RoboDK station: kr30 cnc 070119 wat.rdk

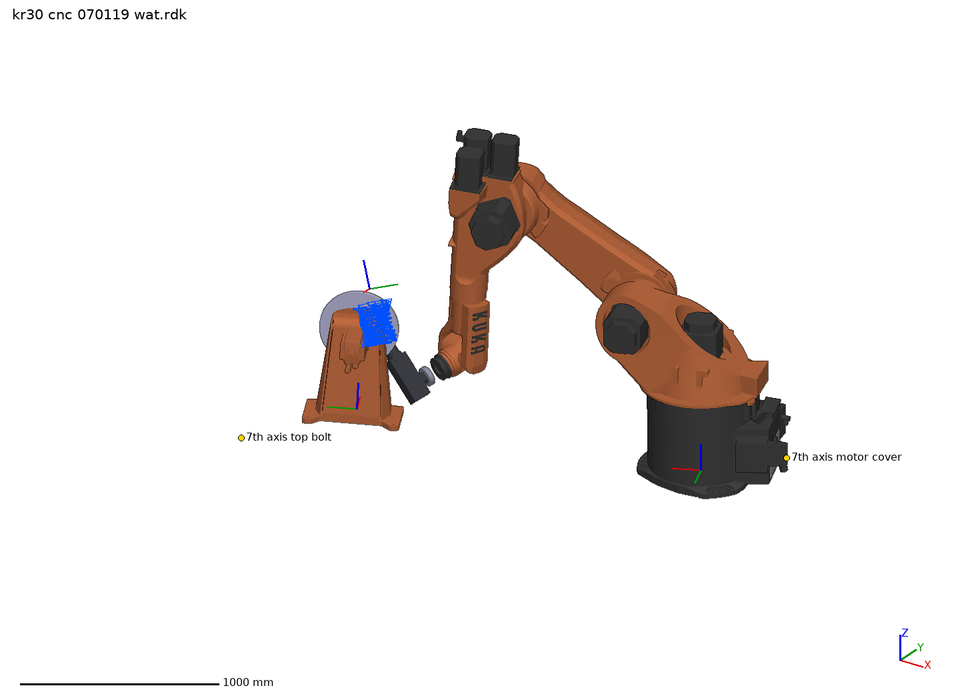
[picture v0: the station drawn from its stored meshes, robots at their saved joint values, targets as dots, program paths as lines]
Station kr30 cnc 070119 wat. Poses are relative to the parent item; angles as X-Y-Z fixed-axis rotations.
  - frame KUKA KR 30 HA Base at (1535.48, 628.29, -1072.61) mm, rotated rx 0 ry 0 rz -156.31 deg
    - robot KUKA KR 30 HA: 6 axes, payload 30 kg, reach 2033 mm, repeatability 0.05 mm, weight 665 kg
        modified DH rows (alpha deg, a mm, theta deg, d mm): 0, 0, 0, 815; -90, 350, 0, 0; 0, 850, -90, 0; -90, 145, 0, 820; 90, 0, 0, 0; -90, 0, 180, 170
        joint limits [-185, -135, -120, -350, -119, -350] to [185, 35, 158, 350, 119, 350]; home [0, -90, 90, 0, 0, 0]; saved at [4.145, -35.537, 122.295, 231.17, 72.258, -40.379]
      - tool 1/2" End Mill TCP, TCP at (337.71, -2.2, 160.57) mm, rotated rx 0 ry 90 rz 0 deg, size 415.8 x 102 x 153.6 mm
    - target 7th axis top bolt (joint target) at (1966.13, 1947.63, 927.26) mm, rotated rx -179.2 ry 6.72 rz -171.11 deg; joints [-17.018, -71.525, 110.046, 168.711, 45.865, -170.331, 883.939] of KUKA KR 30 HA
    - target 7th axis motor cover (joint target) at (-417, -111.35, 57.2) mm, rotated rx -135.46 ry -1.69 rz -48.75 deg; joints [-33.388, -54.543, 96.086, 147.711, 45.276, -113.831, 883.939] of KUKA KR 30 HA
  - frame KUKA KP1 MD250 Base at (172.34, -439.05, -684.5) mm, rotated rx 2 ry 0.52 rz 120.23 deg
    - robot KUKA KP1 MD250: 1 axes, payload 250 kg
        modified DH rows (alpha deg, a mm, theta deg, d mm): 0, 0, 0, 0
        base shift (70, 10, 428) mm, rotated rx 0 ry 90 rz -2 deg
        joint limits [-3600] to [3600]; home [0]; saved at [143.741]
      - frame Frame 2 at (0, 0, 440) mm, rotated rx 0 ry 70 rz 20 deg
  - machining project Machining Settings: C:/Users/liqui/OneDrive/Desktop/suffering.apt | rotz(5) | rotz(80)
  - program Machining (7499 instructions, listed below)
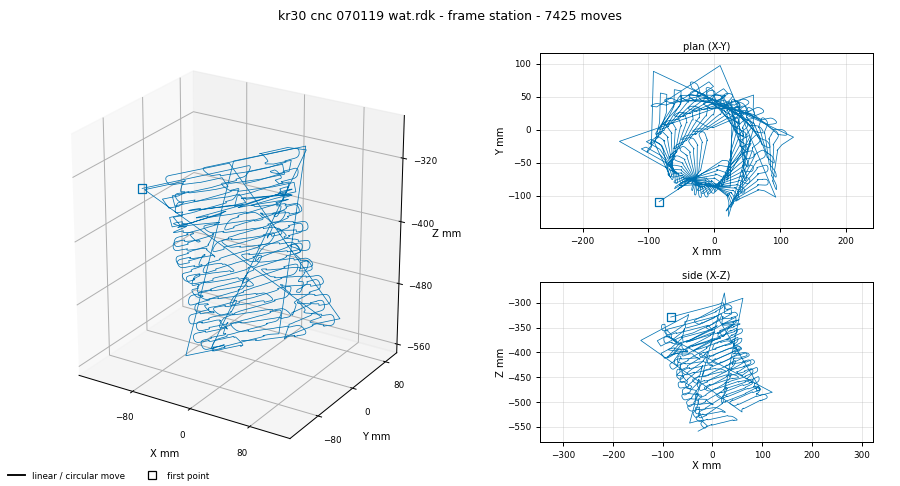
[picture p0: tool path of kr30 cnc 070119 wat.rdk in frame station, 7425 of 7425 moves have a stored position in this frame; points joined in program order, loops and branches not executed]

--- program Machining (robot KUKA KR 30 HA) ---
  Smooth(1)
  Set Ref.: Frame 2
  Set Tool: 1/2" End Mill TCP
  Show 1/2" End Mill TCP
  Print: /'1001'
  Print: /''
  Print: /'Flow1'
  Set speed (1000.0 mm/s)
  Set speed (1000.0 mm/s)
  MoveJ 1 to (78.89, -86.74, -80.36) mm, rotated rx 43.39 ry 15.84 rz 65.61 deg; joints [-0.88, -16.778, 83.729, 155.098, 93.568, 24.647, 178.286]
  MoveL 2 to (78.89, -86.74, -80.36) mm, rotated rx 43.39 ry 15.84 rz 65.61 deg; joints [-0.88, -16.778, 83.729, 155.098, 93.568, 24.647, 178.286]
  MoveL 3 to (78.89, -86.74, -80.36) mm, rotated rx 43.39 ry 15.84 rz 65.61 deg; joints [-0.88, -16.778, 83.729, 155.098, 93.568, 24.647, 178.286]
  Set speed (1000.0 mm/s)
  MoveL 4 to (74.98, -42.03, -80.36) mm, rotated rx 43.39 ry 15.84 rz 65.61 deg; joints [-0.656, -17.28, 87.376, 155.184, 96.389, 23.245, 178.286]
  Set speed (100.0 mm/s)
  MoveL 5 to (68.64, 30.46, -80.36) mm, rotated rx 43.39 ry 15.84 rz 65.61 deg; joints [-0.269, -17.729, 92.84, 155.219, 100.893, 21.011, 178.286]
  MoveL 6 to (68.93, 30.9, -80.36) mm, rotated rx 43.39 ry 15.84 rz 65.61 deg; joints [-0.278, -17.739, 92.882, 155.208, 100.923, 21, 178.286]
  MoveL 7 to (69.23, 31.46, -80.26) mm, rotated rx 43.39 ry 15.84 rz 65.61 deg; joints [-0.286, -17.755, 92.94, 155.197, 100.961, 20.984, 178.286]
  MoveL 8 to (69.53, 31.97, -80.21) mm, rotated rx 43.39 ry 15.84 rz 65.61 deg; joints [-0.294, -17.769, 92.99, 155.187, 100.995, 20.971, 178.286]
  MoveL 9 to (69.83, 32.46, -80.19) mm, rotated rx 43.39 ry 15.84 rz 65.61 deg; joints [-0.303, -17.781, 93.037, 155.176, 101.028, 20.958, 178.286]
  MoveL 10 to (71.83, 35.53, -80.19) mm, rotated rx 43.39 ry 15.84 rz 65.61 deg; joints [-0.366, -17.848, 93.327, 155.099, 101.237, 20.877, 178.286]
  MoveL 11 to (72.67, 36.71, -80.27) mm, rotated rx 43.39 ry 15.84 rz 65.61 deg; joints [-0.394, -17.87, 93.435, 155.066, 101.317, 20.846, 178.286]
  MoveL 12 to (73.47, 37.59, -80.54) mm, rotated rx 43.39 ry 15.84 rz 65.61 deg; joints [-0.423, -17.878, 93.508, 155.033, 101.379, 20.825, 178.286]
  MoveL 13 to (74.21, 38.18, -80.98) mm, rotated rx 43.39 ry 15.84 rz 65.61 deg; joints [-0.455, -17.872, 93.546, 155.001, 101.422, 20.814, 178.286]
  MoveL 14 to (74.56, 38.36, -81.27) mm, rotated rx 43.39 ry 15.84 rz 65.61 deg; joints [-0.471, -17.864, 93.551, 154.985, 101.437, 20.811, 178.286]
  MoveL 15 to (74.9, 38.47, -81.61) mm, rotated rx 43.39 ry 15.84 rz 65.61 deg; joints [-0.487, -17.852, 93.549, 154.969, 101.446, 20.811, 178.286]
  MoveL 16 to (75.55, 38.46, -82.4) mm, rotated rx 43.39 ry 15.84 rz 65.61 deg; joints [-0.521, -17.819, 93.517, 154.937, 101.452, 20.818, 178.286]
  MoveL 17 to (76.14, 38.15, -83.38) mm, rotated rx 43.39 ry 15.84 rz 65.61 deg; joints [-0.557, -17.771, 93.45, 154.906, 101.438, 20.835, 178.286]
  MoveL 18 to (77.19, 36.65, -85.86) mm, rotated rx 43.39 ry 15.84 rz 65.61 deg; joints [-0.633, -17.635, 93.212, 154.845, 101.354, 20.896, 178.286]
  MoveL 19 to (77.76, 34.51, -88.35) mm, rotated rx 43.39 ry 15.84 rz 65.61 deg; joints [-0.693, -17.483, 92.911, 154.802, 101.225, 20.975, 178.286]
  MoveL 20 to (77.59, 32.28, -90.12) mm, rotated rx 43.39 ry 15.84 rz 65.61 deg; joints [-0.717, -17.356, 92.626, 154.793, 101.085, 21.049, 178.286]
  MoveL 21 to (77.22, 31.13, -90.74) mm, rotated rx 43.39 ry 15.84 rz 65.61 deg; joints [-0.715, -17.301, 92.489, 154.801, 101.01, 21.084, 178.286]
  MoveL 22 to (76.67, 29.97, -91.19) mm, rotated rx 43.39 ry 15.84 rz 65.61 deg; joints [-0.705, -17.253, 92.356, 154.818, 100.933, 21.118, 178.286]
  MoveL 23 to (75.02, 27.57, -91.54) mm, rotated rx 43.39 ry 15.84 rz 65.61 deg; joints [-0.657, -17.175, 92.103, 154.876, 100.769, 21.183, 178.286]
  MoveL 24 to (73.01, 25.14, -91.55) mm, rotated rx 43.39 ry 15.84 rz 65.61 deg; joints [-0.593, -17.109, 91.858, 154.95, 100.6, 21.244, 178.286]
  MoveL 25 to (72.71, 24.76, -91.57) mm, rotated rx 43.39 ry 15.84 rz 65.61 deg; joints [-0.583, -17.098, 91.819, 154.96, 100.573, 21.254, 178.286]
  MoveL 26 to (72.43, 24.39, -91.61) mm, rotated rx 43.39 ry 15.84 rz 65.61 deg; joints [-0.575, -17.086, 91.78, 154.97, 100.548, 21.264, 178.286]
  MoveL 27 to (72.2, 24.04, -91.67) mm, rotated rx 43.39 ry 15.84 rz 65.61 deg; joints [-0.569, -17.074, 91.743, 154.978, 100.524, 21.273, 178.286]
  MoveL 28 to (71.94, 23.68, -91.72) mm, rotated rx 43.39 ry 15.84 rz 65.61 deg; joints [-0.561, -17.062, 91.704, 154.987, 100.499, 21.283, 178.286]
  MoveL 29 to (71.6, 23.25, -91.75) mm, rotated rx 43.39 ry 15.84 rz 65.61 deg; joints [-0.551, -17.049, 91.66, 154.999, 100.469, 21.294, 178.286]
  MoveL 30 to (71.2, 22.74, -91.78) mm, rotated rx 43.39 ry 15.84 rz 65.61 deg; joints [-0.539, -17.034, 91.606, 155.013, 100.434, 21.307, 178.286]
  MoveL 31 to (70.87, 22.29, -91.84) mm, rotated rx 43.39 ry 15.84 rz 65.61 deg; joints [-0.529, -17.019, 91.558, 155.025, 100.402, 21.319, 178.286]
  MoveL 32 to (70.62, 21.92, -91.92) mm, rotated rx 43.39 ry 15.84 rz 65.61 deg; joints [-0.522, -17.005, 91.517, 155.033, 100.377, 21.329, 178.286]
  MoveL 33 to (70.37, 21.56, -91.97) mm, rotated rx 43.39 ry 15.84 rz 65.61 deg; joints [-0.515, -16.993, 91.479, 155.042, 100.352, 21.339, 178.286]
  MoveL 34 to (70.07, 21.19, -91.99) mm, rotated rx 43.39 ry 15.84 rz 65.61 deg; joints [-0.506, -16.982, 91.44, 155.052, 100.326, 21.348, 178.286]
  MoveL 35 to (69.74, 20.78, -91.99) mm, rotated rx 43.39 ry 15.84 rz 65.61 deg; joints [-0.495, -16.971, 91.4, 155.064, 100.298, 21.358, 178.286]
  MoveL 36 to (69.39, 20.37, -91.99) mm, rotated rx 43.39 ry 15.84 rz 65.61 deg; joints [-0.484, -16.959, 91.357, 155.077, 100.269, 21.369, 178.286]
  MoveL 37 to (69.04, 19.92, -92) mm, rotated rx 43.39 ry 15.84 rz 65.61 deg; joints [-0.473, -16.947, 91.311, 155.09, 100.238, 21.38, 178.286]
  MoveL 38 to (68.64, 19.39, -92.03) mm, rotated rx 43.39 ry 15.84 rz 65.61 deg; joints [-0.461, -16.931, 91.257, 155.104, 100.201, 21.394, 178.286]
  MoveL 39 to (68.32, 18.89, -92.1) mm, rotated rx 43.39 ry 15.84 rz 65.61 deg; joints [-0.451, -16.915, 91.205, 155.115, 100.167, 21.407, 178.286]
  MoveL 40 to (68.09, 18.5, -92.2) mm, rotated rx 43.39 ry 15.84 rz 65.61 deg; joints [-0.446, -16.9, 91.161, 155.122, 100.14, 21.418, 178.286]
  MoveL 41 to (68.08, 18.51, -92.44) mm, rotated rx 43.39 ry 15.84 rz 65.61 deg; joints [-0.449, -16.885, 91.146, 155.12, 100.14, 21.419, 178.286]
  MoveL 42 to (68.22, 18.88, -92.79) mm, rotated rx 43.39 ry 15.84 rz 65.61 deg; joints [-0.458, -16.869, 91.155, 155.109, 100.165, 21.41, 178.286]
  MoveL 43 to (69.04, 19.11, -93.76) mm, rotated rx 43.39 ry 15.84 rz 65.61 deg; joints [-0.499, -16.831, 91.136, 155.07, 100.186, 21.412, 178.286]
  MoveL 44 to (68.82, 16.99, -93.76) mm, rotated rx 43.39 ry 15.84 rz 65.61 deg; joints [-0.497, -16.812, 90.968, 155.083, 100.051, 21.475, 178.286]
  MoveL 45 to (68.62, 14.7, -93.89) mm, rotated rx 43.39 ry 15.84 rz 65.61 deg; joints [-0.497, -16.783, 90.779, 155.095, 99.906, 21.544, 178.286]
  MoveL 46 to (68.41, 12.54, -93.95) mm, rotated rx 43.39 ry 15.84 rz 65.61 deg; joints [-0.495, -16.759, 90.603, 155.108, 99.768, 21.608, 178.286]
  MoveL 47 to (68.21, 10.42, -94.08) mm, rotated rx 43.39 ry 15.84 rz 65.61 deg; joints [-0.495, -16.731, 90.427, 155.118, 99.634, 21.672, 178.286]
  MoveL 48 to (68.01, 8.29, -94.23) mm, rotated rx 43.39 ry 15.84 rz 65.61 deg; joints [-0.496, -16.7, 90.246, 155.128, 99.498, 21.736, 178.286]
  MoveL 49 to (67.81, 6.18, -94.36) mm, rotated rx 43.39 ry 15.84 rz 65.61 deg; joints [-0.495, -16.671, 90.069, 155.139, 99.363, 21.799, 178.286]
  MoveL 50 to (67.61, 4.04, -94.56) mm, rotated rx 43.39 ry 15.84 rz 65.61 deg; joints [-0.496, -16.637, 89.885, 155.149, 99.227, 21.863, 178.286]
  MoveL 51 to (67.4, 1.93, -94.68) mm, rotated rx 43.39 ry 15.84 rz 65.61 deg; joints [-0.496, -16.608, 89.707, 155.159, 99.092, 21.926, 178.286]
  MoveL 52 to (67.19, -0.21, -94.74) mm, rotated rx 43.39 ry 15.84 rz 65.61 deg; joints [-0.494, -16.582, 89.53, 155.171, 98.955, 21.99, 178.286]
  MoveL 53 to (66.97, -2.35, -94.88) mm, rotated rx 43.39 ry 15.84 rz 65.61 deg; joints [-0.494, -16.549, 89.347, 155.181, 98.818, 22.054, 178.286]
  MoveL 54 to (66.75, -4.57, -95.06) mm, rotated rx 43.39 ry 15.84 rz 65.61 deg; joints [-0.494, -16.514, 89.155, 155.191, 98.676, 22.12, 178.286]
  MoveL 55 to (66.52, -6.78, -95.24) mm, rotated rx 43.39 ry 15.84 rz 65.61 deg; joints [-0.493, -16.478, 88.962, 155.201, 98.534, 22.186, 178.286]
  MoveL 56 to (66.32, -8.65, -95.48) mm, rotated rx 43.39 ry 15.84 rz 65.61 deg; joints [-0.494, -16.441, 88.793, 155.209, 98.414, 22.243, 178.286]
  MoveL 57 to (66.04, -11.3, -95.59) mm, rotated rx 43.39 ry 15.84 rz 65.61 deg; joints [-0.492, -16.403, 88.569, 155.222, 98.244, 22.321, 178.286]
  Set speed (1000.0 mm/s)
  MoveL 58 to (69.99, -56.43, -95.59) mm, rotated rx 43.39 ry 15.84 rz 65.61 deg; joints [-0.725, -16.011, 85.023, 155.17, 95.414, 23.724, 178.286]
  Set speed (1000.0 mm/s)
  MoveL 59 to (64.27, -56.93, -107.47) mm, rotated rx 43.39 ry 15.84 rz 65.61 deg; joints [-0.695, -15.1, 83.995, 155.201, 95.303, 23.764, 178.286]
  Set speed (100.0 mm/s)
  MoveL 60 to (61.77, -28.35, -107.47) mm, rotated rx 43.39 ry 15.84 rz 65.61 deg; joints [-0.549, -15.374, 86.276, 155.242, 97.105, 22.872, 178.286]
  MoveL 61 to (62.19, -26.69, -107.23) mm, rotated rx 43.39 ry 15.84 rz 65.61 deg; joints [-0.556, -15.418, 86.441, 155.23, 97.216, 22.823, 178.286]
  MoveL 62 to (62.63, -24.71, -107.16) mm, rotated rx 43.39 ry 15.84 rz 65.61 deg; joints [-0.565, -15.454, 86.62, 155.213, 97.346, 22.766, 178.286]
  MoveL 63 to (63.09, -22.71, -107.02) mm, rotated rx 43.39 ry 15.84 rz 65.61 deg; joints [-0.574, -15.495, 86.805, 155.197, 97.478, 22.707, 178.286]
  MoveL 64 to (63.66, -20.32, -106.88) mm, rotated rx 43.39 ry 15.84 rz 65.61 deg; joints [-0.586, -15.543, 87.025, 155.176, 97.636, 22.638, 178.286]
  MoveL 65 to (64.13, -18.23, -106.88) mm, rotated rx 43.39 ry 15.84 rz 65.61 deg; joints [-0.598, -15.576, 87.207, 155.158, 97.773, 22.578, 178.286]
  MoveL 66 to (64.64, -15.93, -106.72) mm, rotated rx 43.39 ry 15.84 rz 65.61 deg; joints [-0.608, -15.621, 87.417, 155.139, 97.924, 22.511, 178.286]
  MoveL 67 to (65.09, -13.99, -106.54) mm, rotated rx 43.39 ry 15.84 rz 65.61 deg; joints [-0.616, -15.663, 87.599, 155.123, 98.052, 22.454, 178.286]
  MoveL 68 to (65.55, -12, -106.44) mm, rotated rx 43.39 ry 15.84 rz 65.61 deg; joints [-0.626, -15.699, 87.778, 155.105, 98.183, 22.396, 178.286]
  MoveL 69 to (66.01, -9.91, -106.23) mm, rotated rx 43.39 ry 15.84 rz 65.61 deg; joints [-0.634, -15.744, 87.972, 155.089, 98.32, 22.335, 178.286]
  MoveL 70 to (66.47, -7.85, -106.07) mm, rotated rx 43.39 ry 15.84 rz 65.61 deg; joints [-0.643, -15.784, 88.16, 155.072, 98.455, 22.274, 178.286]
  MoveL 71 to (66.93, -5.79, -105.96) mm, rotated rx 43.39 ry 15.84 rz 65.61 deg; joints [-0.653, -15.821, 88.344, 155.054, 98.589, 22.214, 178.286]
  MoveL 72 to (67.38, -3.69, -105.79) mm, rotated rx 43.39 ry 15.84 rz 65.61 deg; joints [-0.661, -15.861, 88.534, 155.036, 98.726, 22.152, 178.286]
  MoveL 73 to (67.83, -1.62, -105.65) mm, rotated rx 43.39 ry 15.84 rz 65.61 deg; joints [-0.67, -15.899, 88.72, 155.018, 98.862, 22.092, 178.286]
  MoveL 74 to (68.31, 0.51, -105.58) mm, rotated rx 43.39 ry 15.84 rz 65.61 deg; joints [-0.681, -15.933, 88.905, 154.999, 99, 22.03, 178.286]
  MoveL 75 to (68.74, 2.6, -105.38) mm, rotated rx 43.39 ry 15.84 rz 65.61 deg; joints [-0.688, -15.974, 89.095, 154.982, 99.136, 21.968, 178.286]
  MoveL 76 to (69.19, 4.67, -105.25) mm, rotated rx 43.39 ry 15.84 rz 65.61 deg; joints [-0.697, -16.009, 89.278, 154.963, 99.271, 21.907, 178.286]
  MoveL 77 to (69.64, 6.79, -105.13) mm, rotated rx 43.39 ry 15.84 rz 65.61 deg; joints [-0.706, -16.045, 89.464, 154.944, 99.408, 21.845, 178.286]
  MoveL 78 to (69.88, 8.54, -104.92) mm, rotated rx 43.39 ry 15.84 rz 65.61 deg; joints [-0.708, -16.077, 89.621, 154.934, 99.521, 21.792, 178.286]
  MoveL 79 to (69.95, 10.01, -104.57) mm, rotated rx 43.39 ry 15.84 rz 65.61 deg; joints [-0.702, -16.112, 89.76, 154.932, 99.615, 21.746, 178.286]
  MoveL 80 to (69.81, 11.21, -104.04) mm, rotated rx 43.39 ry 15.84 rz 65.61 deg; joints [-0.687, -16.15, 89.882, 154.94, 99.689, 21.706, 178.286]
  MoveL 81 to (69.03, 9.88, -103.19) mm, rotated rx 43.39 ry 15.84 rz 65.61 deg; joints [-0.652, -16.174, 89.813, 154.979, 99.6, 21.737, 178.286]
  MoveL 82 to (69.37, 10.61, -103.19) mm, rotated rx 43.39 ry 15.84 rz 65.61 deg; joints [-0.662, -16.188, 89.879, 154.966, 99.649, 21.717, 178.286]
  MoveL 83 to (69.73, 11.22, -103.19) mm, rotated rx 43.39 ry 15.84 rz 65.61 deg; joints [-0.673, -16.202, 89.937, 154.953, 99.69, 21.701, 178.286]
  MoveL 84 to (70.13, 11.71, -103.18) mm, rotated rx 43.39 ry 15.84 rz 65.61 deg; joints [-0.685, -16.216, 89.988, 154.939, 99.725, 21.688, 178.286]
  MoveL 85 to (70.58, 12.21, -103.16) mm, rotated rx 43.39 ry 15.84 rz 65.61 deg; joints [-0.7, -16.232, 90.041, 154.923, 99.76, 21.676, 178.286]
  MoveL 86 to (71.11, 12.75, -103.13) mm, rotated rx 43.39 ry 15.84 rz 65.61 deg; joints [-0.716, -16.252, 90.102, 154.904, 99.799, 21.663, 178.286]
  MoveL 87 to (72.63, 14.2, -103.13) mm, rotated rx 43.39 ry 15.84 rz 65.61 deg; joints [-0.766, -16.301, 90.26, 154.851, 99.904, 21.628, 178.286]
  MoveL 88 to (72.95, 14.51, -103.11) mm, rotated rx 43.39 ry 15.84 rz 65.61 deg; joints [-0.776, -16.313, 90.295, 154.84, 99.926, 21.621, 178.286]
  MoveL 89 to (73.71, 15.23, -103.11) mm, rotated rx 43.39 ry 15.84 rz 65.61 deg; joints [-0.801, -16.337, 90.374, 154.813, 99.978, 21.603, 178.286]
  MoveL 90 to (74.07, 15.58, -103.1) mm, rotated rx 43.39 ry 15.84 rz 65.61 deg; joints [-0.813, -16.349, 90.412, 154.8, 100.003, 21.595, 178.286]
  MoveL 91 to (74.42, 15.92, -103.08) mm, rotated rx 43.39 ry 15.84 rz 65.61 deg; joints [-0.824, -16.362, 90.45, 154.788, 100.028, 21.587, 178.286]
  MoveL 92 to (74.75, 16.27, -103.05) mm, rotated rx 43.39 ry 15.84 rz 65.61 deg; joints [-0.834, -16.375, 90.489, 154.777, 100.053, 21.578, 178.286]
  MoveL 93 to (75.04, 16.6, -102.99) mm, rotated rx 43.39 ry 15.84 rz 65.61 deg; joints [-0.842, -16.388, 90.527, 154.767, 100.076, 21.57, 178.286]
  MoveL 94 to (75.36, 16.94, -102.96) mm, rotated rx 43.39 ry 15.84 rz 65.61 deg; joints [-0.852, -16.401, 90.566, 154.756, 100.1, 21.561, 178.286]
  MoveL 95 to (75.71, 17.29, -102.94) mm, rotated rx 43.39 ry 15.84 rz 65.61 deg; joints [-0.864, -16.413, 90.604, 154.744, 100.125, 21.552, 178.286]
  MoveL 96 to (76.08, 17.64, -102.93) mm, rotated rx 43.39 ry 15.84 rz 65.61 deg; joints [-0.875, -16.425, 90.643, 154.731, 100.151, 21.544, 178.286]
  MoveL 97 to (76.43, 17.99, -102.91) mm, rotated rx 43.39 ry 15.84 rz 65.61 deg; joints [-0.887, -16.438, 90.682, 154.719, 100.176, 21.535, 178.286]
  MoveL 98 to (76.76, 18.34, -102.87) mm, rotated rx 43.39 ry 15.84 rz 65.61 deg; joints [-0.897, -16.451, 90.721, 154.707, 100.2, 21.527, 178.286]
  MoveL 99 to (77.04, 18.67, -102.82) mm, rotated rx 43.39 ry 15.84 rz 65.61 deg; joints [-0.905, -16.464, 90.758, 154.698, 100.223, 21.518, 178.286]
  MoveL 100 to (77.34, 19.01, -102.76) mm, rotated rx 43.39 ry 15.84 rz 65.61 deg; joints [-0.914, -16.477, 90.797, 154.688, 100.248, 21.509, 178.286]
  MoveL 101 to (78.34, 20.05, -102.68) mm, rotated rx 43.39 ry 15.84 rz 65.61 deg; joints [-0.945, -16.514, 90.912, 154.653, 100.321, 21.483, 178.286]
  MoveL 102 to (79.25, 20.79, -102.81) mm, rotated rx 43.39 ry 15.84 rz 65.61 deg; joints [-0.978, -16.534, 90.988, 154.619, 100.376, 21.467, 178.286]
  MoveL 103 to (80.08, 21.23, -103.15) mm, rotated rx 43.39 ry 15.84 rz 65.61 deg; joints [-1.01, -16.537, 91.025, 154.586, 100.41, 21.46, 178.286]
  MoveL 104 to (80.47, 21.34, -103.39) mm, rotated rx 43.39 ry 15.84 rz 65.61 deg; joints [-1.027, -16.532, 91.029, 154.57, 100.42, 21.46, 178.286]
  MoveL 105 to (80.83, 21.38, -103.69) mm, rotated rx 43.39 ry 15.84 rz 65.61 deg; joints [-1.044, -16.523, 91.023, 154.554, 100.425, 21.463, 178.286]
  MoveL 106 to (81.5, 21.23, -104.45) mm, rotated rx 43.39 ry 15.84 rz 65.61 deg; joints [-1.078, -16.491, 90.982, 154.524, 100.421, 21.475, 178.286]
  MoveL 107 to (82.09, 20.78, -105.42) mm, rotated rx 43.39 ry 15.84 rz 65.61 deg; joints [-1.113, -16.442, 90.902, 154.494, 100.397, 21.497, 178.286]
  MoveL 108 to (83.02, 19, -107.98) mm, rotated rx 43.39 ry 15.84 rz 65.61 deg; joints [-1.184, -16.293, 90.626, 154.438, 100.291, 21.57, 178.286]
  MoveL 109 to (83.37, 16.68, -110.59) mm, rotated rx 43.39 ry 15.84 rz 65.61 deg; joints [-1.237, -16.122, 90.287, 154.403, 100.145, 21.657, 178.286]
  MoveL 110 to (83.23, 15.57, -111.62) mm, rotated rx 43.39 ry 15.84 rz 65.61 deg; joints [-1.249, -16.046, 90.129, 154.399, 100.073, 21.696, 178.286]
  MoveL 111 to (82.89, 14.48, -112.46) mm, rotated rx 43.39 ry 15.84 rz 65.61 deg; joints [-1.25, -15.977, 89.98, 154.403, 100.001, 21.732, 178.286]
  MoveL 112 to (82.34, 13.43, -113.11) mm, rotated rx 43.39 ry 15.84 rz 65.61 deg; joints [-1.242, -15.914, 89.839, 154.417, 99.929, 21.764, 178.286]
  MoveL 113 to (81.58, 12.41, -113.58) mm, rotated rx 43.39 ry 15.84 rz 65.61 deg; joints [-1.224, -15.859, 89.707, 154.439, 99.858, 21.793, 178.286]
  MoveL 114 to (80.61, 11.42, -113.86) mm, rotated rx 43.39 ry 15.84 rz 65.61 deg; joints [-1.197, -15.809, 89.582, 154.47, 99.787, 21.819, 178.286]
  MoveL 115 to (79.44, 10.46, -113.95) mm, rotated rx 43.39 ry 15.84 rz 65.61 deg; joints [-1.159, -15.766, 89.466, 154.51, 99.716, 21.841, 178.286]
  MoveL 116 to (76.9, 8.59, -113.96) mm, rotated rx 43.39 ry 15.84 rz 65.61 deg; joints [-1.075, -15.688, 89.242, 154.597, 99.575, 21.883, 178.286]
  MoveL 117 to (76.46, 8.25, -113.97) mm, rotated rx 43.39 ry 15.84 rz 65.61 deg; joints [-1.061, -15.673, 89.201, 154.612, 99.55, 21.89, 178.286]
  MoveL 118 to (75.97, 7.86, -114.01) mm, rotated rx 43.39 ry 15.84 rz 65.61 deg; joints [-1.045, -15.655, 89.154, 154.629, 99.521, 21.899, 178.286]
  MoveL 119 to (75.4, 7.36, -114.1) mm, rotated rx 43.39 ry 15.84 rz 65.61 deg; joints [-1.028, -15.631, 89.091, 154.647, 99.484, 21.911, 178.286]
  MoveL 120 to (74.92, 6.97, -114.14) mm, rotated rx 43.39 ry 15.84 rz 65.61 deg; joints [-1.012, -15.613, 89.043, 154.664, 99.455, 21.92, 178.286]
  MoveL 121 to (74.49, 6.64, -114.15) mm, rotated rx 43.39 ry 15.84 rz 65.61 deg; joints [-0.998, -15.599, 89.003, 154.678, 99.43, 21.928, 178.286]
  MoveL 122 to (74.08, 6.34, -114.16) mm, rotated rx 43.39 ry 15.84 rz 65.61 deg; joints [-0.985, -15.585, 88.967, 154.692, 99.407, 21.935, 178.286]
  MoveL 123 to (73.72, 6.05, -114.18) mm, rotated rx 43.39 ry 15.84 rz 65.61 deg; joints [-0.974, -15.573, 88.932, 154.704, 99.386, 21.941, 178.286]
  MoveL 124 to (72.07, 4.82, -114.18) mm, rotated rx 43.39 ry 15.84 rz 65.61 deg; joints [-0.919, -15.521, 88.785, 154.76, 99.293, 21.968, 178.286]
  MoveL 125 to (71.67, 4.5, -114.22) mm, rotated rx 43.39 ry 15.84 rz 65.61 deg; joints [-0.907, -15.506, 88.745, 154.774, 99.269, 21.975, 178.286]
  MoveL 126 to (71.32, 4.19, -114.27) mm, rotated rx 43.39 ry 15.84 rz 65.61 deg; joints [-0.896, -15.491, 88.706, 154.785, 99.246, 21.983, 178.286]
  MoveL 127 to (70.98, 3.88, -114.34) mm, rotated rx 43.39 ry 15.84 rz 65.61 deg; joints [-0.886, -15.475, 88.666, 154.796, 99.223, 21.991, 178.286]
  MoveL 128 to (70.64, 3.53, -114.4) mm, rotated rx 43.39 ry 15.84 rz 65.61 deg; joints [-0.876, -15.46, 88.624, 154.807, 99.198, 22, 178.286]
  MoveL 129 to (70.27, 3.12, -114.44) mm, rotated rx 43.39 ry 15.84 rz 65.61 deg; joints [-0.865, -15.445, 88.578, 154.82, 99.169, 22.01, 178.286]
  MoveL 130 to (69.89, 2.57, -114.44) mm, rotated rx 43.39 ry 15.84 rz 65.61 deg; joints [-0.853, -15.43, 88.522, 154.833, 99.13, 22.024, 178.286]
  MoveL 131 to (69.51, 1.89, -114.45) mm, rotated rx 43.39 ry 15.84 rz 65.61 deg; joints [-0.841, -15.415, 88.458, 154.847, 99.084, 22.043, 178.286]
  MoveL 132 to (71.15, 2.93, -116) mm, rotated rx 43.39 ry 15.84 rz 65.61 deg; joints [-0.917, -15.367, 88.486, 154.773, 99.162, 22.03, 178.286]
  MoveL 133 to (70.38, 0.7, -116.13) mm, rotated rx 43.39 ry 15.84 rz 65.61 deg; joints [-0.897, -15.321, 88.279, 154.802, 99.014, 22.094, 178.286]
  MoveL 134 to (69.65, -1.41, -116.24) mm, rotated rx 43.39 ry 15.84 rz 65.61 deg; joints [-0.877, -15.278, 88.083, 154.83, 98.873, 22.154, 178.286]
  MoveL 135 to (68.95, -3.46, -116.4) mm, rotated rx 43.39 ry 15.84 rz 65.61 deg; joints [-0.86, -15.232, 87.89, 154.856, 98.737, 22.213, 178.286]
  MoveL 136 to (68.25, -5.47, -116.51) mm, rotated rx 43.39 ry 15.84 rz 65.61 deg; joints [-0.842, -15.19, 87.702, 154.882, 98.603, 22.271, 178.286]
  MoveL 137 to (67.55, -7.49, -116.62) mm, rotated rx 43.39 ry 15.84 rz 65.61 deg; joints [-0.824, -15.147, 87.513, 154.908, 98.468, 22.329, 178.286]
  MoveL 138 to (66.86, -9.51, -116.84) mm, rotated rx 43.39 ry 15.84 rz 65.61 deg; joints [-0.807, -15.097, 87.316, 154.932, 98.333, 22.387, 178.286]
  MoveL 139 to (66.16, -11.53, -117.07) mm, rotated rx 43.39 ry 15.84 rz 65.61 deg; joints [-0.791, -15.047, 87.119, 154.956, 98.198, 22.445, 178.286]
  MoveL 140 to (65.45, -13.54, -117.18) mm, rotated rx 43.39 ry 15.84 rz 65.61 deg; joints [-0.773, -15.002, 86.928, 154.981, 98.063, 22.503, 178.286]
  MoveL 141 to (64.73, -15.55, -117.18) mm, rotated rx 43.39 ry 15.84 rz 65.61 deg; joints [-0.753, -14.964, 86.745, 155.008, 97.929, 22.559, 178.286]
  MoveL 142 to (64.02, -17.56, -117.29) mm, rotated rx 43.39 ry 15.84 rz 65.61 deg; joints [-0.734, -14.919, 86.553, 155.033, 97.794, 22.616, 178.286]
  MoveL 143 to (63.29, -19.6, -117.5) mm, rotated rx 43.39 ry 15.84 rz 65.61 deg; joints [-0.717, -14.867, 86.352, 155.058, 97.656, 22.675, 178.286]
  MoveL 144 to (62.62, -21.5, -117.67) mm, rotated rx 43.39 ry 15.84 rz 65.61 deg; joints [-0.701, -14.819, 86.166, 155.08, 97.528, 22.729, 178.286]
  MoveL 145 to (61.99, -23.25, -117.89) mm, rotated rx 43.39 ry 15.84 rz 65.61 deg; joints [-0.686, -14.772, 85.99, 155.1, 97.41, 22.779, 178.286]
  MoveL 146 to (61.33, -25.1, -117.98) mm, rotated rx 43.39 ry 15.84 rz 65.61 deg; joints [-0.669, -14.729, 85.812, 155.123, 97.285, 22.831, 178.286]
  MoveL 147 to (60.62, -27.07, -117.99) mm, rotated rx 43.39 ry 15.84 rz 65.61 deg; joints [-0.65, -14.689, 85.629, 155.148, 97.152, 22.886, 178.286]
  MoveL 148 to (59.7, -29.61, -118.09) mm, rotated rx 43.39 ry 15.84 rz 65.61 deg; joints [-0.625, -14.631, 85.384, 155.18, 96.98, 22.958, 178.286]
  MoveL 149 to (58.99, -31.52, -118.3) mm, rotated rx 43.39 ry 15.84 rz 65.61 deg; joints [-0.609, -14.578, 85.191, 155.202, 96.85, 23.012, 178.286]
  MoveL 150 to (58.22, -33.58, -118.51) mm, rotated rx 43.39 ry 15.84 rz 65.61 deg; joints [-0.59, -14.522, 84.983, 155.227, 96.709, 23.071, 178.286]
  MoveL 151 to (57.5, -35.47, -118.79) mm, rotated rx 43.39 ry 15.84 rz 65.61 deg; joints [-0.574, -14.464, 84.784, 155.248, 96.58, 23.125, 178.286]
  MoveL 152 to (56.82, -37.34, -118.92) mm, rotated rx 43.39 ry 15.84 rz 65.61 deg; joints [-0.557, -14.416, 84.599, 155.27, 96.453, 23.178, 178.286]
  MoveL 153 to (56.11, -39.31, -118.94) mm, rotated rx 43.39 ry 15.84 rz 65.61 deg; joints [-0.538, -14.373, 84.412, 155.294, 96.319, 23.233, 178.286]
  MoveL 154 to (55.46, -40.96, -119.17) mm, rotated rx 43.39 ry 15.84 rz 65.61 deg; joints [-0.523, -14.322, 84.238, 155.313, 96.205, 23.279, 178.286]
  Set speed (1000.0 mm/s)
  MoveL 155 to (57.74, -66.91, -119.17) mm, rotated rx 43.39 ry 15.84 rz 65.61 deg; joints [-0.655, -14.043, 82.122, 155.266, 94.556, 24.094, 178.286]
  Set speed (1000.0 mm/s)
  MoveL 156 to (51.22, -67.48, -130.35) mm, rotated rx 43.39 ry 15.84 rz 65.61 deg; joints [-0.591, -13.142, 81.063, 155.33, 94.403, 24.138, 178.286]
  Set speed (100.0 mm/s)
  MoveL 157 to (49.47, -47.39, -130.35) mm, rotated rx 43.39 ry 15.84 rz 65.61 deg; joints [-0.488, -13.368, 82.718, 155.369, 95.685, 23.506, 178.286]
  MoveL 158 to (50.43, -45.49, -130.35) mm, rotated rx 43.39 ry 15.84 rz 65.61 deg; joints [-0.516, -13.418, 82.911, 155.338, 95.819, 23.455, 178.286]
  MoveL 159 to (51.46, -43.51, -130.25) mm, rotated rx 43.39 ry 15.84 rz 65.61 deg; joints [-0.545, -13.476, 83.118, 155.306, 95.959, 23.401, 178.286]
  MoveL 160 to (52.58, -41.44, -129.96) mm, rotated rx 43.39 ry 15.84 rz 65.61 deg; joints [-0.573, -13.55, 83.349, 155.273, 96.106, 23.344, 178.286]
  MoveL 161 to (53.65, -39.46, -129.62) mm, rotated rx 43.39 ry 15.84 rz 65.61 deg; joints [-0.6, -13.624, 83.574, 155.242, 96.247, 23.289, 178.286]
  MoveL 162 to (54.61, -37.63, -129.43) mm, rotated rx 43.39 ry 15.84 rz 65.61 deg; joints [-0.625, -13.684, 83.771, 155.213, 96.376, 23.239, 178.286]
  MoveL 163 to (55.5, -35.9, -129.29) mm, rotated rx 43.39 ry 15.84 rz 65.61 deg; joints [-0.65, -13.736, 83.954, 155.185, 96.498, 23.191, 178.286]
  MoveL 164 to (56.44, -34.07, -129.24) mm, rotated rx 43.39 ry 15.84 rz 65.61 deg; joints [-0.676, -13.785, 84.14, 155.154, 96.625, 23.142, 178.286]
  MoveL 165 to (57.4, -32.17, -129.22) mm, rotated rx 43.39 ry 15.84 rz 65.61 deg; joints [-0.704, -13.834, 84.33, 155.122, 96.758, 23.09, 178.286]
  MoveL 166 to (58.36, -30.28, -129.1) mm, rotated rx 43.39 ry 15.84 rz 65.61 deg; joints [-0.731, -13.887, 84.525, 155.091, 96.89, 23.039, 178.286]
  MoveL 167 to (59.41, -28.24, -128.84) mm, rotated rx 43.39 ry 15.84 rz 65.61 deg; joints [-0.758, -13.954, 84.744, 155.058, 97.032, 22.982, 178.286]
  MoveL 168 to (60.49, -26.1, -128.66) mm, rotated rx 43.39 ry 15.84 rz 65.61 deg; joints [-0.787, -14.017, 84.968, 155.023, 97.181, 22.923, 178.286]
  MoveL 169 to (61.54, -24.01, -128.45) mm, rotated rx 43.39 ry 15.84 rz 65.61 deg; joints [-0.815, -14.079, 85.185, 154.989, 97.326, 22.865, 178.286]
  MoveL 170 to (62.5, -22.11, -128.34) mm, rotated rx 43.39 ry 15.84 rz 65.61 deg; joints [-0.842, -14.131, 85.379, 154.957, 97.458, 22.812, 178.286]
  MoveL 171 to (64.38, -18.33, -128.07) mm, rotated rx 43.39 ry 15.84 rz 65.61 deg; joints [-0.894, -14.236, 85.764, 154.894, 97.719, 22.708, 178.286]
  MoveL 172 to (65.36, -16.38, -128) mm, rotated rx 43.39 ry 15.84 rz 65.61 deg; joints [-0.923, -14.285, 85.957, 154.86, 97.853, 22.654, 178.286]
  MoveL 173 to (66.3, -14.47, -127.78) mm, rotated rx 43.39 ry 15.84 rz 65.61 deg; joints [-0.947, -14.342, 86.156, 154.829, 97.985, 22.6, 178.286]
  MoveL 174 to (67.23, -12.57, -127.62) mm, rotated rx 43.39 ry 15.84 rz 65.61 deg; joints [-0.973, -14.394, 86.348, 154.797, 98.115, 22.547, 178.286]
  MoveL 175 to (68.15, -10.67, -127.44) mm, rotated rx 43.39 ry 15.84 rz 65.61 deg; joints [-0.998, -14.448, 86.542, 154.766, 98.245, 22.494, 178.286]
  MoveL 176 to (69.12, -8.72, -127.34) mm, rotated rx 43.39 ry 15.84 rz 65.61 deg; joints [-1.026, -14.496, 86.734, 154.731, 98.378, 22.44, 178.286]
  MoveL 177 to (70.11, -6.68, -127.22) mm, rotated rx 43.39 ry 15.84 rz 65.61 deg; joints [-1.054, -14.548, 86.936, 154.696, 98.518, 22.383, 178.286]
  MoveL 178 to (70.97, -4.98, -127.16) mm, rotated rx 43.39 ry 15.84 rz 65.61 deg; joints [-1.079, -14.589, 87.102, 154.665, 98.634, 22.336, 178.286]
  MoveL 179 to (70.38, -4.68, -126.27) mm, rotated rx 43.39 ry 15.84 rz 65.61 deg; joints [-1.046, -14.633, 87.167, 154.694, 98.649, 22.318, 178.286]
  MoveL 180 to (70.06, -4.84, -125.86) mm, rotated rx 43.39 ry 15.84 rz 65.61 deg; joints [-1.03, -14.65, 87.173, 154.709, 98.637, 22.318, 178.286]
  MoveL 181 to (69.99, -4.83, -125.58) mm, rotated rx 43.39 ry 15.84 rz 65.61 deg; joints [-1.024, -14.666, 87.19, 154.715, 98.638, 22.315, 178.286]
  MoveL 182 to (70.25, -4.63, -125.46) mm, rotated rx 43.39 ry 15.84 rz 65.61 deg; joints [-1.031, -14.681, 87.222, 154.707, 98.654, 22.31, 178.286]
  MoveL 183 to (70.62, -4.38, -125.4) mm, rotated rx 43.39 ry 15.84 rz 65.61 deg; joints [-1.042, -14.697, 87.258, 154.696, 98.673, 22.305, 178.286]
  MoveL 184 to (71.1, -4.08, -125.37) mm, rotated rx 43.39 ry 15.84 rz 65.61 deg; joints [-1.057, -14.714, 87.299, 154.68, 98.697, 22.298, 178.286]
  MoveL 185 to (71.69, -3.72, -125.33) mm, rotated rx 43.39 ry 15.84 rz 65.61 deg; joints [-1.076, -14.735, 87.349, 154.661, 98.726, 22.291, 178.286]
  MoveL 186 to (72.24, -3.4, -125.31) mm, rotated rx 43.39 ry 15.84 rz 65.61 deg; joints [-1.094, -14.753, 87.394, 154.643, 98.751, 22.285, 178.286]
  MoveL 187 to (72.69, -3.14, -125.31) mm, rotated rx 43.39 ry 15.84 rz 65.61 deg; joints [-1.109, -14.767, 87.428, 154.628, 98.772, 22.28, 178.286]
  MoveL 188 to (73.12, -2.89, -125.29) mm, rotated rx 43.39 ry 15.84 rz 65.61 deg; joints [-1.123, -14.781, 87.462, 154.614, 98.792, 22.275, 178.286]
  MoveL 189 to (73.99, -2.34, -125.21) mm, rotated rx 43.39 ry 15.84 rz 65.61 deg; joints [-1.151, -14.814, 87.539, 154.586, 98.836, 22.263, 178.286]
  MoveL 190 to (74.47, -2.03, -125.16) mm, rotated rx 43.39 ry 15.84 rz 65.61 deg; joints [-1.166, -14.831, 87.581, 154.57, 98.859, 22.257, 178.286]
  MoveL 191 to (74.88, -1.74, -125.09) mm, rotated rx 43.39 ry 15.84 rz 65.61 deg; joints [-1.178, -14.849, 87.622, 154.557, 98.882, 22.25, 178.286]
  MoveL 192 to (75.26, -1.47, -125.02) mm, rotated rx 43.39 ry 15.84 rz 65.61 deg; joints [-1.19, -14.866, 87.66, 154.545, 98.903, 22.244, 178.286]
  MoveL 193 to (75.65, -1.22, -124.96) mm, rotated rx 43.39 ry 15.84 rz 65.61 deg; joints [-1.202, -14.881, 87.696, 154.533, 98.923, 22.238, 178.286]
  MoveL 194 to (76.06, -0.96, -124.93) mm, rotated rx 43.39 ry 15.84 rz 65.61 deg; joints [-1.215, -14.896, 87.732, 154.52, 98.943, 22.233, 178.286]
  MoveL 195 to (76.51, -0.69, -124.91) mm, rotated rx 43.39 ry 15.84 rz 65.61 deg; joints [-1.23, -14.911, 87.768, 154.505, 98.964, 22.227, 178.286]
  MoveL 196 to (79.7, 1.1, -124.91) mm, rotated rx 43.39 ry 15.84 rz 65.61 deg; joints [-1.336, -15.008, 88.008, 154.398, 99.107, 22.193, 178.286]
  MoveL 197 to (81.17, 1.8, -124.93) mm, rotated rx 43.39 ry 15.84 rz 65.61 deg; joints [-1.385, -15.05, 88.107, 154.349, 99.165, 22.181, 178.286]
  MoveL 198 to (81.72, 1.97, -124.96) mm, rotated rx 43.39 ry 15.84 rz 65.61 deg; joints [-1.404, -15.063, 88.135, 154.33, 99.18, 22.18, 178.286]
  MoveL 199 to (82.16, 2.01, -124.99) mm, rotated rx 43.39 ry 15.84 rz 65.61 deg; joints [-1.42, -15.073, 88.15, 154.316, 99.187, 22.182, 178.286]
  MoveL 200 to (82.5, 1.96, -125.03) mm, rotated rx 43.39 ry 15.84 rz 65.61 deg; joints [-1.432, -15.078, 88.153, 154.305, 99.187, 22.186, 178.286]
  MoveL 201 to (82.63, 1.89, -125.06) mm, rotated rx 43.39 ry 15.84 rz 65.61 deg; joints [-1.437, -15.08, 88.151, 154.3, 99.184, 22.189, 178.286]
  MoveL 202 to (82.74, 1.81, -125.08) mm, rotated rx 43.39 ry 15.84 rz 65.61 deg; joints [-1.441, -15.08, 88.146, 154.297, 99.179, 22.193, 178.286]
  MoveL 203 to (82.83, 1.7, -125.11) mm, rotated rx 43.39 ry 15.84 rz 65.61 deg; joints [-1.445, -15.08, 88.139, 154.294, 99.173, 22.197, 178.286]
  MoveL 204 to (82.9, 1.58, -125.14) mm, rotated rx 43.39 ry 15.84 rz 65.61 deg; joints [-1.448, -15.079, 88.129, 154.292, 99.166, 22.201, 178.286]
  MoveL 205 to (82.98, 1.27, -125.2) mm, rotated rx 43.39 ry 15.84 rz 65.61 deg; joints [-1.452, -15.075, 88.103, 154.29, 99.147, 22.212, 178.286]
  MoveL 206 to (82.93, 0.48, -125.33) mm, rotated rx 43.39 ry 15.84 rz 65.61 deg; joints [-1.453, -15.059, 88.031, 154.292, 99.097, 22.237, 178.286]
  MoveL 207 to (82.67, -0.5, -125.47) mm, rotated rx 43.39 ry 15.84 rz 65.61 deg; joints [-1.448, -15.035, 87.938, 154.302, 99.033, 22.266, 178.286]
  MoveL 208 to (81.78, -2.66, -125.74) mm, rotated rx 43.39 ry 15.84 rz 65.61 deg; joints [-1.425, -14.977, 87.722, 154.334, 98.888, 22.329, 178.286]
  MoveL 209 to (80.71, -4.82, -125.98) mm, rotated rx 43.39 ry 15.84 rz 65.61 deg; joints [-1.395, -14.916, 87.502, 154.372, 98.741, 22.391, 178.286]
  MoveL 210 to (56.48, -53.07, -131.06) mm, rotated rx 43.39 ry 15.84 rz 65.61 deg; joints [-0.742, -13.437, 82.427, 155.155, 95.397, 23.739, 178.286]
  MoveL 211 to (54.76, -56.49, -131.42) mm, rotated rx 43.39 ry 15.84 rz 65.61 deg; joints [-0.697, -13.322, 82.052, 155.205, 95.154, 23.834, 178.286]
  MoveL 212 to (52.92, -59.76, -131.84) mm, rotated rx 43.39 ry 15.84 rz 65.61 deg; joints [-0.649, -13.201, 81.681, 155.258, 94.92, 23.923, 178.286]
  MoveL 213 to (51.96, -60.9, -132.05) mm, rotated rx 43.39 ry 15.84 rz 65.61 deg; joints [-0.623, -13.146, 81.536, 155.285, 94.833, 23.953, 178.286]
  MoveL 214 to (51.51, -61.2, -132.15) mm, rotated rx 43.39 ry 15.84 rz 65.61 deg; joints [-0.61, -13.124, 81.487, 155.298, 94.808, 23.959, 178.286]
  MoveL 215 to (51.29, -61.27, -132.19) mm, rotated rx 43.39 ry 15.84 rz 65.61 deg; joints [-0.604, -13.114, 81.471, 155.304, 94.8, 23.96, 178.286]
  MoveL 216 to (51.08, -61.28, -132.23) mm, rotated rx 43.39 ry 15.84 rz 65.61 deg; joints [-0.597, -13.106, 81.46, 155.309, 94.797, 23.959, 178.286]
  MoveL 217 to (50.88, -61.21, -132.27) mm, rotated rx 43.39 ry 15.84 rz 65.61 deg; joints [-0.591, -13.099, 81.456, 155.315, 94.799, 23.955, 178.286]
  MoveL 218 to (50.69, -61.08, -132.3) mm, rotated rx 43.39 ry 15.84 rz 65.61 deg; joints [-0.585, -13.094, 81.459, 155.32, 94.806, 23.95, 178.286]
  MoveL 219 to (50.52, -60.86, -132.33) mm, rotated rx 43.39 ry 15.84 rz 65.61 deg; joints [-0.579, -13.09, 81.469, 155.325, 94.817, 23.942, 178.286]
  MoveL 220 to (50.35, -60.56, -132.36) mm, rotated rx 43.39 ry 15.84 rz 65.61 deg; joints [-0.573, -13.088, 81.487, 155.329, 94.835, 23.932, 178.286]
  MoveL 221 to (49.85, -58.43, -132.41) mm, rotated rx 43.39 ry 15.84 rz 65.61 deg; joints [-0.553, -13.101, 81.65, 155.342, 94.967, 23.862, 178.286]
  MoveL 222 to (49.6, -56.35, -132.41) mm, rotated rx 43.39 ry 15.84 rz 65.61 deg; joints [-0.54, -13.123, 81.819, 155.349, 95.099, 23.796, 178.286]
  MoveL 223 to (49.6, -52.55, -132.45) mm, rotated rx 43.39 ry 15.84 rz 65.61 deg; joints [-0.532, -13.171, 82.139, 155.345, 95.345, 23.68, 178.286]
  MoveL 224 to (50.37, -49.09, -132.56) mm, rotated rx 43.39 ry 15.84 rz 65.61 deg; joints [-0.551, -13.229, 82.45, 155.318, 95.578, 23.58, 178.286]
  MoveL 225 to (53.08, -43.68, -132.86) mm, rotated rx 43.39 ry 15.84 rz 65.61 deg; joints [-0.634, -13.35, 82.975, 155.226, 95.957, 23.437, 178.286]
  MoveL 226 to (54.56, -41.83, -132.99) mm, rotated rx 43.39 ry 15.84 rz 65.61 deg; joints [-0.68, -13.404, 83.17, 155.178, 96.092, 23.392, 178.286]
  MoveL 227 to (77.42, -15.64, -134.86) mm, rotated rx 43.39 ry 15.84 rz 65.61 deg; joints [-1.422, -14.168, 85.928, 154.4, 98, 22.759, 178.286]
  MoveL 228 to (79.36, -13.39, -135.02) mm, rotated rx 43.39 ry 15.84 rz 65.61 deg; joints [-1.487, -14.229, 86.158, 154.331, 98.161, 22.704, 178.286]
  MoveL 229 to (81.44, -10.29, -135.26) mm, rotated rx 43.39 ry 15.84 rz 65.61 deg; joints [-1.555, -14.296, 86.453, 154.254, 98.376, 22.623, 178.286]
  MoveL 230 to (81.98, -8.9, -135.4) mm, rotated rx 43.39 ry 15.84 rz 65.61 deg; joints [-1.573, -14.313, 86.57, 154.231, 98.468, 22.584, 178.286]
  MoveL 231 to (82.01, -8.36, -135.47) mm, rotated rx 43.39 ry 15.84 rz 65.61 deg; joints [-1.574, -14.315, 86.61, 154.227, 98.502, 22.567, 178.286]
  MoveL 232 to (81.96, -8.14, -135.51) mm, rotated rx 43.39 ry 15.84 rz 65.61 deg; joints [-1.573, -14.313, 86.623, 154.228, 98.516, 22.56, 178.286]
  MoveL 233 to (81.86, -7.95, -135.54) mm, rotated rx 43.39 ry 15.84 rz 65.61 deg; joints [-1.57, -14.31, 86.632, 154.23, 98.526, 22.554, 178.286]
  MoveL 234 to (81.7, -7.81, -135.58) mm, rotated rx 43.39 ry 15.84 rz 65.61 deg; joints [-1.564, -14.305, 86.636, 154.234, 98.533, 22.549, 178.286]
  MoveL 235 to (81.49, -7.72, -135.61) mm, rotated rx 43.39 ry 15.84 rz 65.61 deg; joints [-1.557, -14.298, 86.634, 154.24, 98.537, 22.545, 178.286]
  MoveL 236 to (81.21, -7.67, -135.64) mm, rotated rx 43.39 ry 15.84 rz 65.61 deg; joints [-1.548, -14.289, 86.627, 154.248, 98.537, 22.542, 178.286]
  MoveL 237 to (80.87, -7.68, -135.68) mm, rotated rx 43.39 ry 15.84 rz 65.61 deg; joints [-1.537, -14.278, 86.613, 154.259, 98.533, 22.54, 178.286]
  MoveL 238 to (78.78, -8.34, -135.8) mm, rotated rx 43.39 ry 15.84 rz 65.61 deg; joints [-1.469, -14.211, 86.486, 154.325, 98.471, 22.547, 178.286]
  MoveL 239 to (78.3, -8.55, -135.82) mm, rotated rx 43.39 ry 15.84 rz 65.61 deg; joints [-1.453, -14.195, 86.454, 154.34, 98.453, 22.55, 178.286]
  MoveL 240 to (77.89, -8.76, -135.87) mm, rotated rx 43.39 ry 15.84 rz 65.61 deg; joints [-1.44, -14.18, 86.421, 154.353, 98.436, 22.554, 178.286]
  MoveL 241 to (77.51, -8.97, -135.94) mm, rotated rx 43.39 ry 15.84 rz 65.61 deg; joints [-1.428, -14.163, 86.386, 154.365, 98.418, 22.558, 178.286]
  MoveL 242 to (77.11, -9.18, -136) mm, rotated rx 43.39 ry 15.84 rz 65.61 deg; joints [-1.416, -14.148, 86.354, 154.378, 98.401, 22.562, 178.286]
  MoveL 243 to (76.7, -9.38, -136.03) mm, rotated rx 43.39 ry 15.84 rz 65.61 deg; joints [-1.403, -14.133, 86.322, 154.391, 98.384, 22.566, 178.286]
  MoveL 244 to (72.36, -11.14, -136.04) mm, rotated rx 43.39 ry 15.84 rz 65.61 deg; joints [-1.258, -14.004, 86.043, 154.532, 98.23, 22.591, 178.286]
  MoveL 245 to (71.95, -11.32, -136.06) mm, rotated rx 43.39 ry 15.84 rz 65.61 deg; joints [-1.245, -13.991, 86.014, 154.545, 98.214, 22.594, 178.286]
  MoveL 246 to (71.51, -11.51, -136.08) mm, rotated rx 43.39 ry 15.84 rz 65.61 deg; joints [-1.231, -13.977, 85.985, 154.559, 98.198, 22.597, 178.286]
  MoveL 247 to (70.55, -11.9, -136.08) mm, rotated rx 43.39 ry 15.84 rz 65.61 deg; joints [-1.199, -13.948, 85.922, 154.59, 98.163, 22.602, 178.286]
  MoveL 248 to (70.03, -12.12, -136.08) mm, rotated rx 43.39 ry 15.84 rz 65.61 deg; joints [-1.182, -13.932, 85.887, 154.607, 98.144, 22.606, 178.286]
  MoveL 249 to (69.48, -12.38, -136.1) mm, rotated rx 43.39 ry 15.84 rz 65.61 deg; joints [-1.164, -13.914, 85.848, 154.624, 98.122, 22.61, 178.286]
  MoveL 250 to (68.9, -12.69, -136.13) mm, rotated rx 43.39 ry 15.84 rz 65.61 deg; joints [-1.145, -13.894, 85.802, 154.643, 98.096, 22.616, 178.286]
  MoveL 251 to (68.36, -13.07, -136.15) mm, rotated rx 43.39 ry 15.84 rz 65.61 deg; joints [-1.128, -13.875, 85.752, 154.661, 98.066, 22.624, 178.286]
  MoveL 252 to (67.85, -13.49, -136.17) mm, rotated rx 43.39 ry 15.84 rz 65.61 deg; joints [-1.112, -13.857, 85.701, 154.677, 98.034, 22.634, 178.286]
  MoveL 253 to (69.02, -12.9, -137.15) mm, rotated rx 43.39 ry 15.84 rz 65.61 deg; joints [-1.164, -13.831, 85.718, 154.627, 98.081, 22.63, 178.286]
  MoveL 254 to (68.56, -14.15, -137.58) mm, rotated rx 43.39 ry 15.84 rz 65.61 deg; joints [-1.156, -13.779, 85.573, 154.64, 97.994, 22.668, 178.286]
  MoveL 255 to (67.92, -15.5, -137.9) mm, rotated rx 43.39 ry 15.84 rz 65.61 deg; joints [-1.141, -13.729, 85.422, 154.66, 97.901, 22.708, 178.286]
  MoveL 256 to (67.08, -16.98, -138.13) mm, rotated rx 43.39 ry 15.84 rz 65.61 deg; joints [-1.119, -13.678, 85.26, 154.686, 97.798, 22.749, 178.286]
  MoveL 257 to (65.93, -18.77, -138.35) mm, rotated rx 43.39 ry 15.84 rz 65.61 deg; joints [-1.086, -13.616, 85.062, 154.724, 97.671, 22.799, 178.286]
  MoveL 258 to (64.75, -20.55, -138.46) mm, rotated rx 43.39 ry 15.84 rz 65.61 deg; joints [-1.052, -13.56, 84.872, 154.763, 97.545, 22.846, 178.286]
  MoveL 259 to (63.57, -22.33, -138.57) mm, rotated rx 43.39 ry 15.84 rz 65.61 deg; joints [-1.017, -13.504, 84.681, 154.802, 97.418, 22.894, 178.286]
  MoveL 260 to (62.4, -24.12, -138.8) mm, rotated rx 43.39 ry 15.84 rz 65.61 deg; joints [-0.984, -13.44, 84.481, 154.839, 97.291, 22.942, 178.286]
  MoveL 261 to (61.22, -25.89, -138.92) mm, rotated rx 43.39 ry 15.84 rz 65.61 deg; joints [-0.949, -13.382, 84.29, 154.878, 97.164, 22.99, 178.286]
  MoveL 262 to (60.04, -27.67, -139.15) mm, rotated rx 43.39 ry 15.84 rz 65.61 deg; joints [-0.917, -13.317, 84.089, 154.915, 97.037, 23.038, 178.286]
  MoveL 263 to (58.85, -29.44, -139.27) mm, rotated rx 43.39 ry 15.84 rz 65.61 deg; joints [-0.882, -13.259, 83.896, 154.954, 96.91, 23.085, 178.286]
  MoveL 264 to (57.66, -31.21, -139.39) mm, rotated rx 43.39 ry 15.84 rz 65.61 deg; joints [-0.847, -13.2, 83.702, 154.992, 96.783, 23.132, 178.286]
  MoveL 265 to (56.47, -32.98, -139.62) mm, rotated rx 43.39 ry 15.84 rz 65.61 deg; joints [-0.814, -13.134, 83.5, 155.029, 96.655, 23.179, 178.286]
  MoveL 266 to (55.32, -34.67, -139.73) mm, rotated rx 43.39 ry 15.84 rz 65.61 deg; joints [-0.781, -13.077, 83.314, 155.065, 96.534, 23.224, 178.286]
  MoveL 267 to (54.19, -36.3, -139.93) mm, rotated rx 43.39 ry 15.84 rz 65.61 deg; joints [-0.749, -13.015, 83.126, 155.1, 96.415, 23.268, 178.286]
  MoveL 268 to (52.87, -38.27, -140.09) mm, rotated rx 43.39 ry 15.84 rz 65.61 deg; joints [-0.711, -12.946, 82.906, 155.141, 96.272, 23.32, 178.286]
  MoveL 269 to (51.31, -40.51, -140.18) mm, rotated rx 43.39 ry 15.84 rz 65.61 deg; joints [-0.666, -12.872, 82.661, 155.19, 96.11, 23.378, 178.286]
  MoveL 270 to (50.15, -42.23, -140.25) mm, rotated rx 43.39 ry 15.84 rz 65.61 deg; joints [-0.632, -12.816, 82.473, 155.227, 95.985, 23.423, 178.286]
  MoveL 271 to (49.07, -43.82, -140.38) mm, rotated rx 43.39 ry 15.84 rz 65.61 deg; joints [-0.601, -12.759, 82.293, 155.26, 95.869, 23.465, 178.286]
  MoveL 272 to (47.95, -45.46, -140.48) mm, rotated rx 43.39 ry 15.84 rz 65.61 deg; joints [-0.569, -12.702, 82.109, 155.294, 95.75, 23.507, 178.286]
  MoveL 273 to (46.84, -47.06, -140.59) mm, rotated rx 43.39 ry 15.84 rz 65.61 deg; joints [-0.537, -12.644, 81.927, 155.328, 95.632, 23.55, 178.286]
  MoveL 274 to (45.68, -48.77, -140.66) mm, rotated rx 43.39 ry 15.84 rz 65.61 deg; joints [-0.504, -12.587, 81.739, 155.364, 95.508, 23.594, 178.286]
  MoveL 275 to (44.42, -50.6, -140.76) mm, rotated rx 43.39 ry 15.84 rz 65.61 deg; joints [-0.467, -12.523, 81.532, 155.402, 95.373, 23.641, 178.286]
  MoveL 276 to (43.02, -52.56, -141.02) mm, rotated rx 43.39 ry 15.84 rz 65.61 deg; joints [-0.429, -12.442, 81.298, 155.442, 95.228, 23.693, 178.286]
  MoveL 277 to (42.2, -54.64, -142.01) mm, rotated rx 43.39 ry 15.84 rz 65.61 deg; joints [-0.42, -12.328, 81.021, 155.457, 95.078, 23.758, 178.286]
  MoveL 278 to (42.21, -53.5, -142.49) mm, rotated rx 43.39 ry 15.84 rz 65.61 deg; joints [-0.424, -12.313, 81.083, 155.45, 95.15, 23.727, 178.286]
  MoveL 279 to (42.22, -52.9, -142.8) mm, rotated rx 43.39 ry 15.84 rz 65.61 deg; joints [-0.427, -12.301, 81.112, 155.446, 95.187, 23.711, 178.286]
  MoveL 280 to (42.21, -52.8, -142.95) mm, rotated rx 43.39 ry 15.84 rz 65.61 deg; joints [-0.429, -12.292, 81.11, 155.444, 95.193, 23.709, 178.286]
  MoveL 281 to (42.21, -53.15, -142.99) mm, rotated rx 43.39 ry 15.84 rz 65.61 deg; joints [-0.43, -12.285, 81.077, 155.444, 95.17, 23.72, 178.286]
  MoveL 282 to (42.2, -53.61, -143.01) mm, rotated rx 43.39 ry 15.84 rz 65.61 deg; joints [-0.431, -12.278, 81.036, 155.445, 95.139, 23.734, 178.286]
  MoveL 283 to (42.17, -54.09, -143.04) mm, rotated rx 43.39 ry 15.84 rz 65.61 deg; joints [-0.432, -12.268, 80.992, 155.445, 95.108, 23.749, 178.286]
  MoveL 284 to (42.14, -54.54, -143.1) mm, rotated rx 43.39 ry 15.84 rz 65.61 deg; joints [-0.432, -12.257, 80.948, 155.446, 95.078, 23.763, 178.286]
  MoveL 285 to (42.11, -55, -143.14) mm, rotated rx 43.39 ry 15.84 rz 65.61 deg; joints [-0.433, -12.248, 80.904, 155.447, 95.047, 23.777, 178.286]
  MoveL 286 to (42.1, -55.49, -143.16) mm, rotated rx 43.39 ry 15.84 rz 65.61 deg; joints [-0.434, -12.239, 80.86, 155.447, 95.015, 23.792, 178.286]
  MoveL 287 to (42.08, -58.11, -143.16) mm, rotated rx 43.39 ry 15.84 rz 65.61 deg; joints [-0.439, -12.203, 80.635, 155.449, 94.844, 23.873, 178.286]
  MoveL 288 to (42.07, -58.57, -143.18) mm, rotated rx 43.39 ry 15.84 rz 65.61 deg; joints [-0.44, -12.195, 80.594, 155.449, 94.814, 23.887, 178.286]
  MoveL 289 to (42.04, -58.96, -143.21) mm, rotated rx 43.39 ry 15.84 rz 65.61 deg; joints [-0.441, -12.186, 80.557, 155.45, 94.788, 23.899, 178.286]
  MoveL 290 to (42.03, -59.42, -143.24) mm, rotated rx 43.39 ry 15.84 rz 65.61 deg; joints [-0.441, -12.178, 80.515, 155.45, 94.758, 23.913, 178.286]
  MoveL 291 to (42.01, -60.01, -143.26) mm, rotated rx 43.39 ry 15.84 rz 65.61 deg; joints [-0.443, -12.168, 80.462, 155.451, 94.719, 23.932, 178.286]
  MoveL 292 to (41.97, -60.74, -143.31) mm, rotated rx 43.39 ry 15.84 rz 65.61 deg; joints [-0.443, -12.153, 80.394, 155.452, 94.671, 23.954, 178.286]
  MoveL 293 to (41.94, -61.35, -143.34) mm, rotated rx 43.39 ry 15.84 rz 65.61 deg; joints [-0.444, -12.142, 80.338, 155.452, 94.63, 23.973, 178.286]
  MoveL 294 to (41.94, -61.89, -143.34) mm, rotated rx 43.39 ry 15.84 rz 65.61 deg; joints [-0.446, -12.134, 80.291, 155.453, 94.595, 23.99, 178.286]
  MoveL 295 to (41.93, -63.46, -143.34) mm, rotated rx 43.39 ry 15.84 rz 65.61 deg; joints [-0.449, -12.111, 80.155, 155.454, 94.492, 24.038, 178.286]
  MoveL 296 to (41.62, -66.35, -143.68) mm, rotated rx 43.39 ry 15.84 rz 65.61 deg; joints [-0.45, -12.038, 79.867, 155.46, 94.297, 24.128, 178.286]
  MoveL 297 to (41.25, -67.6, -144.11) mm, rotated rx 43.39 ry 15.84 rz 65.61 deg; joints [-0.446, -11.982, 79.714, 155.466, 94.209, 24.167, 178.286]
  MoveL 298 to (40.73, -68.7, -144.71) mm, rotated rx 43.39 ry 15.84 rz 65.61 deg; joints [-0.439, -11.912, 79.556, 155.475, 94.127, 24.202, 178.286]
  MoveL 299 to (39.25, -70.49, -146.42) mm, rotated rx 43.39 ry 15.84 rz 65.61 deg; joints [-0.418, -11.734, 79.221, 155.499, 93.981, 24.259, 178.286]
  MoveL 300 to (37.18, -71.72, -148.82) mm, rotated rx 43.39 ry 15.84 rz 65.61 deg; joints [-0.385, -11.502, 78.862, 155.532, 93.859, 24.301, 178.286]
  MoveL 301 to (35.17, -72.16, -151.21) mm, rotated rx 43.39 ry 15.84 rz 65.61 deg; joints [-0.352, -11.284, 78.573, 155.563, 93.79, 24.318, 178.286]
  MoveL 302 to (34.43, -72, -152.16) mm, rotated rx 43.39 ry 15.84 rz 65.61 deg; joints [-0.34, -11.205, 78.491, 155.574, 93.785, 24.315, 178.286]
  MoveL 303 to (33.86, -71.58, -152.93) mm, rotated rx 43.39 ry 15.84 rz 65.61 deg; joints [-0.33, -11.146, 78.45, 155.582, 93.8, 24.304, 178.286]
  MoveL 304 to (33.63, -71.27, -153.25) mm, rotated rx 43.39 ry 15.84 rz 65.61 deg; joints [-0.327, -11.123, 78.445, 155.585, 93.815, 24.296, 178.286]
  MoveL 305 to (33.46, -70.9, -153.52) mm, rotated rx 43.39 ry 15.84 rz 65.61 deg; joints [-0.324, -11.106, 78.45, 155.587, 93.836, 24.285, 178.286]
  MoveL 306 to (33.23, -69.97, -153.95) mm, rotated rx 43.39 ry 15.84 rz 65.61 deg; joints [-0.32, -11.086, 78.493, 155.589, 93.892, 24.258, 178.286]
  MoveL 307 to (33.18, -68.78, -154.21) mm, rotated rx 43.39 ry 15.84 rz 65.61 deg; joints [-0.319, -11.087, 78.577, 155.587, 93.968, 24.223, 178.286]
  MoveL 308 to (33.3, -67.34, -154.29) mm, rotated rx 43.39 ry 15.84 rz 65.61 deg; joints [-0.321, -11.106, 78.702, 155.583, 94.064, 24.18, 178.286]
  MoveL 309 to (33.37, -66.82, -154.29) mm, rotated rx 43.39 ry 15.84 rz 65.61 deg; joints [-0.322, -11.116, 78.75, 155.581, 94.099, 24.165, 178.286]
  MoveL 310 to (33.47, -66.39, -154.24) mm, rotated rx 43.39 ry 15.84 rz 65.61 deg; joints [-0.323, -11.129, 78.795, 155.579, 94.129, 24.152, 178.286]
  MoveL 311 to (33.57, -65.97, -154.18) mm, rotated rx 43.39 ry 15.84 rz 65.61 deg; joints [-0.325, -11.142, 78.84, 155.576, 94.159, 24.139, 178.286]
  MoveL 312 to (33.66, -65.5, -154.14) mm, rotated rx 43.39 ry 15.84 rz 65.61 deg; joints [-0.326, -11.154, 78.887, 155.574, 94.191, 24.125, 178.286]
  MoveL 313 to (33.73, -65.01, -154.12) mm, rotated rx 43.39 ry 15.84 rz 65.61 deg; joints [-0.327, -11.164, 78.934, 155.572, 94.224, 24.11, 178.286]
  MoveL 314 to (33.81, -64.48, -154.12) mm, rotated rx 43.39 ry 15.84 rz 65.61 deg; joints [-0.328, -11.175, 78.984, 155.57, 94.26, 24.094, 178.286]
  MoveL 315 to (33.88, -63.96, -154.12) mm, rotated rx 43.39 ry 15.84 rz 65.61 deg; joints [-0.329, -11.184, 79.032, 155.567, 94.295, 24.079, 178.286]
  MoveL 316 to (33.93, -63.46, -154.13) mm, rotated rx 43.39 ry 15.84 rz 65.61 deg; joints [-0.33, -11.192, 79.077, 155.566, 94.329, 24.064, 178.286]
  MoveL 317 to (33.99, -62.97, -154.15) mm, rotated rx 43.39 ry 15.84 rz 65.61 deg; joints [-0.331, -11.2, 79.121, 155.564, 94.362, 24.049, 178.286]
  MoveL 318 to (34.06, -62.51, -154.13) mm, rotated rx 43.39 ry 15.84 rz 65.61 deg; joints [-0.332, -11.21, 79.165, 155.562, 94.393, 24.035, 178.286]
  MoveL 319 to (34.14, -62.05, -154.09) mm, rotated rx 43.39 ry 15.84 rz 65.61 deg; joints [-0.333, -11.222, 79.211, 155.56, 94.424, 24.021, 178.286]
  MoveL 320 to (34.25, -61.52, -154.04) mm, rotated rx 43.39 ry 15.84 rz 65.61 deg; joints [-0.335, -11.236, 79.265, 155.557, 94.461, 24.005, 178.286]
  MoveL 321 to (34.39, -60.83, -153.98) mm, rotated rx 43.39 ry 15.84 rz 65.61 deg; joints [-0.337, -11.253, 79.334, 155.553, 94.508, 23.985, 178.286]
  MoveL 322 to (34.49, -60.19, -153.96) mm, rotated rx 43.39 ry 15.84 rz 65.61 deg; joints [-0.339, -11.267, 79.395, 155.55, 94.552, 23.966, 178.286]
  MoveL 323 to (34.84, -57.6, -153.96) mm, rotated rx 43.39 ry 15.84 rz 65.61 deg; joints [-0.344, -11.313, 79.632, 155.539, 94.726, 23.888, 178.286]
  MoveL 324 to (34.94, -56.98, -153.92) mm, rotated rx 43.39 ry 15.84 rz 65.61 deg; joints [-0.345, -11.327, 79.692, 155.536, 94.768, 23.87, 178.286]
  MoveL 325 to (35.04, -56.43, -153.86) mm, rotated rx 43.39 ry 15.84 rz 65.61 deg; joints [-0.346, -11.341, 79.747, 155.534, 94.806, 23.853, 178.286]
  MoveL 326 to (35.08, -56.23, -153.71) mm, rotated rx 43.39 ry 15.84 rz 65.61 deg; joints [-0.345, -11.355, 79.777, 155.534, 94.82, 23.846, 178.286]
  MoveL 327 to (35.06, -56.35, -153.45) mm, rotated rx 43.39 ry 15.84 rz 65.61 deg; joints [-0.341, -11.37, 79.785, 155.538, 94.814, 23.847, 178.286]
  MoveL 328 to (34.97, -56.79, -153.05) mm, rotated rx 43.39 ry 15.84 rz 65.61 deg; joints [-0.334, -11.387, 79.773, 155.545, 94.786, 23.857, 178.286]
  MoveL 329 to (35.98, -56.6, -152.24) mm, rotated rx 43.39 ry 15.84 rz 65.61 deg; joints [-0.356, -11.47, 79.885, 155.525, 94.816, 23.852, 178.286]
  MoveL 330 to (37.33, -55.16, -152.02) mm, rotated rx 43.39 ry 15.84 rz 65.61 deg; joints [-0.394, -11.541, 80.074, 155.486, 94.929, 23.816, 178.286]
  MoveL 331 to (38.68, -53.68, -151.87) mm, rotated rx 43.39 ry 15.84 rz 65.61 deg; joints [-0.433, -11.608, 80.261, 155.447, 95.044, 23.779, 178.286]
  MoveL 332 to (40.06, -52.15, -151.71) mm, rotated rx 43.39 ry 15.84 rz 65.61 deg; joints [-0.473, -11.676, 80.452, 155.406, 95.162, 23.741, 178.286]
  MoveL 333 to (41.33, -50.77, -151.42) mm, rotated rx 43.39 ry 15.84 rz 65.61 deg; joints [-0.508, -11.748, 80.637, 155.37, 95.269, 23.705, 178.286]
  MoveL 334 to (42.75, -49.2, -151.23) mm, rotated rx 43.39 ry 15.84 rz 65.61 deg; joints [-0.548, -11.82, 80.834, 155.329, 95.39, 23.666, 178.286]
  MoveL 335 to (44.23, -47.56, -151.05) mm, rotated rx 43.39 ry 15.84 rz 65.61 deg; joints [-0.591, -11.893, 81.039, 155.285, 95.516, 23.625, 178.286]
  MoveL 336 to (45.73, -45.89, -150.96) mm, rotated rx 43.39 ry 15.84 rz 65.61 deg; joints [-0.636, -11.961, 81.239, 155.239, 95.643, 23.583, 178.286]
  MoveL 337 to (47.54, -43.85, -150.87) mm, rotated rx 43.39 ry 15.84 rz 65.61 deg; joints [-0.69, -12.041, 81.481, 155.183, 95.797, 23.533, 178.286]
  MoveL 338 to (48.84, -42.38, -150.77) mm, rotated rx 43.39 ry 15.84 rz 65.61 deg; joints [-0.729, -12.101, 81.657, 155.144, 95.908, 23.496, 178.286]
  MoveL 339 to (50.05, -41.01, -150.55) mm, rotated rx 43.39 ry 15.84 rz 65.61 deg; joints [-0.763, -12.164, 81.83, 155.108, 96.012, 23.461, 178.286]
  MoveL 340 to (51.38, -39.5, -150.36) mm, rotated rx 43.39 ry 15.84 rz 65.61 deg; joints [-0.802, -12.231, 82.016, 155.067, 96.127, 23.422, 178.286]
  MoveL 341 to (52.79, -37.9, -150.24) mm, rotated rx 43.39 ry 15.84 rz 65.61 deg; joints [-0.844, -12.296, 82.207, 155.024, 96.247, 23.382, 178.286]
  MoveL 342 to (54.18, -36.3, -150.06) mm, rotated rx 43.39 ry 15.84 rz 65.61 deg; joints [-0.884, -12.363, 82.4, 154.981, 96.367, 23.341, 178.286]
  MoveL 343 to (55.57, -34.71, -149.94) mm, rotated rx 43.39 ry 15.84 rz 65.61 deg; joints [-0.926, -12.427, 82.588, 154.937, 96.486, 23.301, 178.286]
  MoveL 344 to (57, -33.07, -149.76) mm, rotated rx 43.39 ry 15.84 rz 65.61 deg; joints [-0.968, -12.495, 82.786, 154.893, 96.609, 23.259, 178.286]
  MoveL 345 to (58.4, -31.46, -149.64) mm, rotated rx 43.39 ry 15.84 rz 65.61 deg; joints [-1.01, -12.558, 82.974, 154.849, 96.728, 23.218, 178.286]
  MoveL 346 to (59.79, -29.83, -149.41) mm, rotated rx 43.39 ry 15.84 rz 65.61 deg; joints [-1.05, -12.628, 83.172, 154.806, 96.849, 23.175, 178.286]
  MoveL 347 to (61.19, -28.22, -149.3) mm, rotated rx 43.39 ry 15.84 rz 65.61 deg; joints [-1.092, -12.69, 83.359, 154.761, 96.969, 23.134, 178.286]
  MoveL 348 to (62.58, -26.6, -149.18) mm, rotated rx 43.39 ry 15.84 rz 65.61 deg; joints [-1.134, -12.752, 83.547, 154.717, 97.088, 23.093, 178.286]
  MoveL 349 to (63.96, -24.97, -148.96) mm, rotated rx 43.39 ry 15.84 rz 65.61 deg; joints [-1.174, -12.82, 83.742, 154.673, 97.209, 23.05, 178.286]
  MoveL 350 to (65.17, -23.46, -148.76) mm, rotated rx 43.39 ry 15.84 rz 65.61 deg; joints [-1.209, -12.881, 83.92, 154.635, 97.32, 23.01, 178.286]
  MoveL 351 to (66.22, -22.04, -148.46) mm, rotated rx 43.39 ry 15.84 rz 65.61 deg; joints [-1.238, -12.942, 84.09, 154.603, 97.423, 22.971, 178.286]
  MoveL 352 to (67.13, -20.68, -148.06) mm, rotated rx 43.39 ry 15.84 rz 65.61 deg; joints [-1.261, -13.006, 84.259, 154.576, 97.521, 22.932, 178.286]
  MoveL 353 to (65.81, -21.39, -147.13) mm, rotated rx 43.39 ry 15.84 rz 65.61 deg; joints [-1.205, -13.024, 84.225, 154.63, 97.466, 22.939, 178.286]
  MoveL 354 to (66.28, -21.04, -147.12) mm, rotated rx 43.39 ry 15.84 rz 65.61 deg; joints [-1.22, -13.04, 84.269, 154.615, 97.493, 22.931, 178.286]
  MoveL 355 to (66.72, -20.75, -147.1) mm, rotated rx 43.39 ry 15.84 rz 65.61 deg; joints [-1.234, -13.056, 84.309, 154.6, 97.516, 22.925, 178.286]
  MoveL 356 to (67.14, -20.53, -147.04) mm, rotated rx 43.39 ry 15.84 rz 65.61 deg; joints [-1.247, -13.073, 84.345, 154.588, 97.535, 22.921, 178.286]
  MoveL 357 to (67.54, -20.34, -146.97) mm, rotated rx 43.39 ry 15.84 rz 65.61 deg; joints [-1.26, -13.09, 84.378, 154.575, 97.552, 22.917, 178.286]
  MoveL 358 to (67.98, -20.18, -146.92) mm, rotated rx 43.39 ry 15.84 rz 65.61 deg; joints [-1.273, -13.106, 84.409, 154.562, 97.567, 22.915, 178.286]
  MoveL 359 to (68.44, -20.03, -146.89) mm, rotated rx 43.39 ry 15.84 rz 65.61 deg; joints [-1.288, -13.122, 84.438, 154.548, 97.581, 22.913, 178.286]
  MoveL 360 to (68.95, -19.89, -146.87) mm, rotated rx 43.39 ry 15.84 rz 65.61 deg; joints [-1.305, -13.138, 84.468, 154.532, 97.596, 22.912, 178.286]
  MoveL 361 to (69.46, -19.75, -146.87) mm, rotated rx 43.39 ry 15.84 rz 65.61 deg; joints [-1.322, -13.152, 84.495, 154.516, 97.61, 22.912, 178.286]
  MoveL 362 to (69.91, -19.62, -146.86) mm, rotated rx 43.39 ry 15.84 rz 65.61 deg; joints [-1.336, -13.166, 84.521, 154.502, 97.623, 22.91, 178.286]
  MoveL 363 to (70.31, -19.49, -146.84) mm, rotated rx 43.39 ry 15.84 rz 65.61 deg; joints [-1.349, -13.179, 84.546, 154.489, 97.636, 22.909, 178.286]
  MoveL 364 to (70.77, -19.36, -146.82) mm, rotated rx 43.39 ry 15.84 rz 65.61 deg; joints [-1.365, -13.194, 84.573, 154.475, 97.649, 22.908, 178.286]
  MoveL 365 to (71.28, -19.23, -146.82) mm, rotated rx 43.39 ry 15.84 rz 65.61 deg; joints [-1.381, -13.208, 84.601, 154.459, 97.663, 22.907, 178.286]
  MoveL 366 to (71.87, -19.06, -146.8) mm, rotated rx 43.39 ry 15.84 rz 65.61 deg; joints [-1.401, -13.227, 84.635, 154.44, 97.68, 22.906, 178.286]
  MoveL 367 to (72.53, -18.86, -146.76) mm, rotated rx 43.39 ry 15.84 rz 65.61 deg; joints [-1.422, -13.249, 84.675, 154.419, 97.699, 22.904, 178.286]
  MoveL 368 to (73.12, -18.7, -146.74) mm, rotated rx 43.39 ry 15.84 rz 65.61 deg; joints [-1.442, -13.267, 84.709, 154.401, 97.716, 22.903, 178.286]
  MoveL 369 to (73.73, -18.51, -146.71) mm, rotated rx 43.39 ry 15.84 rz 65.61 deg; joints [-1.462, -13.286, 84.745, 154.382, 97.734, 22.902, 178.286]
  MoveL 370 to (74.41, -18.3, -146.68) mm, rotated rx 43.39 ry 15.84 rz 65.61 deg; joints [-1.484, -13.308, 84.787, 154.361, 97.755, 22.899, 178.286]
  MoveL 371 to (74.98, -18.14, -146.66) mm, rotated rx 43.39 ry 15.84 rz 65.61 deg; joints [-1.502, -13.325, 84.819, 154.343, 97.771, 22.898, 178.286]
  MoveL 372 to (75.51, -18, -146.66) mm, rotated rx 43.39 ry 15.84 rz 65.61 deg; joints [-1.52, -13.341, 84.848, 154.326, 97.785, 22.898, 178.286]
  MoveL 373 to (77.03, -17.6, -146.66) mm, rotated rx 43.39 ry 15.84 rz 65.61 deg; joints [-1.571, -13.384, 84.929, 154.278, 97.826, 22.896, 178.286]
  MoveL 374 to (78.45, -17.3, -146.74) mm, rotated rx 43.39 ry 15.84 rz 65.61 deg; joints [-1.619, -13.418, 84.992, 154.232, 97.859, 22.897, 178.286]
  MoveL 375 to (79.63, -17.2, -147) mm, rotated rx 43.39 ry 15.84 rz 65.61 deg; joints [-1.663, -13.433, 85.02, 154.192, 97.876, 22.904, 178.286]
  MoveL 376 to (80.58, -17.3, -147.42) mm, rotated rx 43.39 ry 15.84 rz 65.61 deg; joints [-1.701, -13.43, 85.012, 154.157, 97.877, 22.917, 178.286]
  MoveL 377 to (80.97, -17.43, -147.69) mm, rotated rx 43.39 ry 15.84 rz 65.61 deg; joints [-1.718, -13.421, 84.994, 154.142, 97.872, 22.925, 178.286]
  MoveL 378 to (81.3, -17.61, -148.01) mm, rotated rx 43.39 ry 15.84 rz 65.61 deg; joints [-1.733, -13.407, 84.968, 154.129, 97.862, 22.936, 178.286]
  MoveL 379 to (81.79, -18.13, -148.77) mm, rotated rx 43.39 ry 15.84 rz 65.61 deg; joints [-1.761, -13.366, 84.888, 154.106, 97.831, 22.961, 178.286]
  MoveL 380 to (82.04, -18.84, -149.7) mm, rotated rx 43.39 ry 15.84 rz 65.61 deg; joints [-1.783, -13.306, 84.772, 154.09, 97.784, 22.991, 178.286]
  MoveL 381 to (81.84, -20.89, -152.06) mm, rotated rx 43.39 ry 15.84 rz 65.61 deg; joints [-1.81, -13.128, 84.431, 154.074, 97.642, 23.071, 178.286]
  MoveL 382 to (80.86, -23.09, -154.42) mm, rotated rx 43.39 ry 15.84 rz 65.61 deg; joints [-1.812, -12.928, 84.052, 154.083, 97.481, 23.151, 178.286]
  MoveL 383 to (79.27, -24.78, -156.11) mm, rotated rx 43.39 ry 15.84 rz 65.61 deg; joints [-1.783, -12.761, 83.742, 154.117, 97.349, 23.205, 178.286]
  MoveL 384 to (78.24, -25.43, -156.7) mm, rotated rx 43.39 ry 15.84 rz 65.61 deg; joints [-1.757, -12.689, 83.613, 154.144, 97.294, 23.222, 178.286]
  MoveL 385 to (77.05, -25.95, -157.12) mm, rotated rx 43.39 ry 15.84 rz 65.61 deg; joints [-1.724, -12.625, 83.502, 154.177, 97.246, 23.234, 178.286]
  MoveL 386 to (74.21, -26.62, -157.46) mm, rotated rx 43.39 ry 15.84 rz 65.61 deg; joints [-1.634, -12.523, 83.331, 154.262, 97.172, 23.237, 178.286]
  MoveL 387 to (70.06, -27.15, -157.46) mm, rotated rx 43.39 ry 15.84 rz 65.61 deg; joints [-1.496, -12.409, 83.152, 154.391, 97.093, 23.224, 178.286]
  MoveL 388 to (69.51, -27.24, -157.48) mm, rotated rx 43.39 ry 15.84 rz 65.61 deg; joints [-1.478, -12.392, 83.125, 154.408, 97.082, 23.223, 178.286]
  MoveL 389 to (68.99, -27.33, -157.52) mm, rotated rx 43.39 ry 15.84 rz 65.61 deg; joints [-1.461, -12.375, 83.098, 154.424, 97.07, 23.222, 178.286]
  MoveL 390 to (68.48, -27.44, -157.58) mm, rotated rx 43.39 ry 15.84 rz 65.61 deg; joints [-1.445, -12.356, 83.067, 154.439, 97.057, 23.223, 178.286]
  MoveL 391 to (67.97, -27.57, -157.66) mm, rotated rx 43.39 ry 15.84 rz 65.61 deg; joints [-1.429, -12.336, 83.034, 154.454, 97.043, 23.224, 178.286]
  MoveL 392 to (67.48, -27.69, -157.74) mm, rotated rx 43.39 ry 15.84 rz 65.61 deg; joints [-1.414, -12.317, 83.002, 154.468, 97.029, 23.224, 178.286]
  MoveL 393 to (67, -27.78, -157.78) mm, rotated rx 43.39 ry 15.84 rz 65.61 deg; joints [-1.399, -12.301, 82.977, 154.483, 97.018, 23.224, 178.286]
  MoveL 394 to (66.53, -27.85, -157.8) mm, rotated rx 43.39 ry 15.84 rz 65.61 deg; joints [-1.383, -12.287, 82.954, 154.497, 97.008, 23.223, 178.286]
  MoveL 395 to (66.01, -27.92, -157.8) mm, rotated rx 43.39 ry 15.84 rz 65.61 deg; joints [-1.366, -12.272, 82.931, 154.513, 96.998, 23.222, 178.286]
  MoveL 396 to (65.39, -28.02, -157.83) mm, rotated rx 43.39 ry 15.84 rz 65.61 deg; joints [-1.346, -12.253, 82.9, 154.532, 96.985, 23.221, 178.286]
  MoveL 397 to (64.72, -28.14, -157.89) mm, rotated rx 43.39 ry 15.84 rz 65.61 deg; joints [-1.324, -12.23, 82.863, 154.552, 96.969, 23.22, 178.286]
  MoveL 398 to (64.14, -28.26, -157.91) mm, rotated rx 43.39 ry 15.84 rz 65.61 deg; joints [-1.305, -12.212, 82.832, 154.57, 96.955, 23.22, 178.286]
  MoveL 399 to (63.6, -28.4, -157.92) mm, rotated rx 43.39 ry 15.84 rz 65.61 deg; joints [-1.288, -12.196, 82.802, 154.587, 96.94, 23.221, 178.286]
  MoveL 400 to (63.08, -28.6, -157.92) mm, rotated rx 43.39 ry 15.84 rz 65.61 deg; joints [-1.271, -12.18, 82.769, 154.603, 96.921, 23.223, 178.286]
  MoveL 401 to (62.59, -28.9, -157.92) mm, rotated rx 43.39 ry 15.84 rz 65.61 deg; joints [-1.255, -12.164, 82.727, 154.619, 96.896, 23.229, 178.286]
  MoveL 402 to (62.11, -29.29, -157.92) mm, rotated rx 43.39 ry 15.84 rz 65.61 deg; joints [-1.24, -12.147, 82.679, 154.634, 96.867, 23.238, 178.286]
  MoveL 403 to (63.53, -28.6, -158.88) mm, rotated rx 43.39 ry 15.84 rz 65.61 deg; joints [-1.299, -12.13, 82.714, 154.578, 96.921, 23.234, 178.286]
  MoveL 404 to (62.76, -29.58, -159.3) mm, rotated rx 43.39 ry 15.84 rz 65.61 deg; joints [-1.28, -12.071, 82.576, 154.599, 96.847, 23.262, 178.286]
  MoveL 405 to (61.81, -30.63, -159.63) mm, rotated rx 43.39 ry 15.84 rz 65.61 deg; joints [-1.255, -12.013, 82.434, 154.627, 96.767, 23.291, 178.286]
  MoveL 406 to (60.67, -31.76, -159.88) mm, rotated rx 43.39 ry 15.84 rz 65.61 deg; joints [-1.222, -11.954, 82.283, 154.661, 96.68, 23.32, 178.286]
  MoveL 407 to (59.08, -33.19, -159.99) mm, rotated rx 43.39 ry 15.84 rz 65.61 deg; joints [-1.173, -11.888, 82.104, 154.711, 96.57, 23.354, 178.286]
  MoveL 408 to (57.51, -34.62, -160.22) mm, rotated rx 43.39 ry 15.84 rz 65.61 deg; joints [-1.126, -11.815, 81.914, 154.759, 96.458, 23.39, 178.286]
  MoveL 409 to (55.92, -36.04, -160.34) mm, rotated rx 43.39 ry 15.84 rz 65.61 deg; joints [-1.078, -11.748, 81.733, 154.808, 96.348, 23.424, 178.286]
  MoveL 410 to (54.32, -37.46, -160.45) mm, rotated rx 43.39 ry 15.84 rz 65.61 deg; joints [-1.029, -11.681, 81.551, 154.858, 96.237, 23.458, 178.286]
  MoveL 411 to (52.74, -38.89, -160.69) mm, rotated rx 43.39 ry 15.84 rz 65.61 deg; joints [-0.982, -11.607, 81.36, 154.905, 96.124, 23.492, 178.286]
  MoveL 412 to (51.14, -40.3, -160.81) mm, rotated rx 43.39 ry 15.84 rz 65.61 deg; joints [-0.934, -11.539, 81.177, 154.954, 96.013, 23.526, 178.286]
  MoveL 413 to (49.54, -41.71, -160.93) mm, rotated rx 43.39 ry 15.84 rz 65.61 deg; joints [-0.885, -11.471, 80.994, 155.003, 95.902, 23.56, 178.286]
  MoveL 414 to (47.7, -43.34, -161.08) mm, rotated rx 43.39 ry 15.84 rz 65.61 deg; joints [-0.83, -11.39, 80.781, 155.059, 95.773, 23.598, 178.286]
  MoveL 415 to (46.12, -44.73, -161.28) mm, rotated rx 43.39 ry 15.84 rz 65.61 deg; joints [-0.783, -11.317, 80.594, 155.106, 95.663, 23.632, 178.286]
  MoveL 416 to (44.38, -46.25, -161.48) mm, rotated rx 43.39 ry 15.84 rz 65.61 deg; joints [-0.732, -11.238, 80.389, 155.158, 95.541, 23.668, 178.286]
  MoveL 417 to (42.68, -47.73, -161.73) mm, rotated rx 43.39 ry 15.84 rz 65.61 deg; joints [-0.682, -11.156, 80.184, 155.208, 95.422, 23.704, 178.286]
  MoveL 418 to (41.07, -49.13, -161.85) mm, rotated rx 43.39 ry 15.84 rz 65.61 deg; joints [-0.634, -11.086, 79.998, 155.256, 95.309, 23.737, 178.286]
  MoveL 419 to (39.46, -50.54, -161.85) mm, rotated rx 43.39 ry 15.84 rz 65.61 deg; joints [-0.584, -11.023, 79.82, 155.305, 95.197, 23.769, 178.286]
  MoveL 420 to (37.87, -51.92, -161.93) mm, rotated rx 43.39 ry 15.84 rz 65.61 deg; joints [-0.536, -10.956, 79.639, 155.353, 95.087, 23.8, 178.286]
  MoveL 421 to (36.31, -53.25, -162.14) mm, rotated rx 43.39 ry 15.84 rz 65.61 deg; joints [-0.49, -10.881, 79.452, 155.398, 94.978, 23.832, 178.286]
  MoveL 422 to (34.54, -54.73, -162.49) mm, rotated rx 43.39 ry 15.84 rz 65.61 deg; joints [-0.44, -10.79, 79.235, 155.448, 94.856, 23.868, 178.286]
  MoveL 423 to (33.15, -55.89, -162.71) mm, rotated rx 43.39 ry 15.84 rz 65.61 deg; joints [-0.4, -10.721, 79.068, 155.487, 94.76, 23.895, 178.286]
  MoveL 424 to (31.25, -57.44, -163) mm, rotated rx 43.39 ry 15.84 rz 65.61 deg; joints [-0.346, -10.628, 78.842, 155.541, 94.631, 23.932, 178.286]
  MoveL 425 to (29.57, -58.88, -163.11) mm, rotated rx 43.39 ry 15.84 rz 65.61 deg; joints [-0.296, -10.554, 78.648, 155.59, 94.514, 23.965, 178.286]
  MoveL 426 to (27.97, -60.27, -163.12) mm, rotated rx 43.39 ry 15.84 rz 65.61 deg; joints [-0.247, -10.489, 78.466, 155.638, 94.4, 23.997, 178.286]
  MoveL 427 to (27.08, -60.39, -163.91) mm, rotated rx 43.39 ry 15.84 rz 65.61 deg; joints [-0.229, -10.411, 78.364, 155.655, 94.375, 24.001, 178.286]
  MoveL 428 to (27.27, -59.99, -164.3) mm, rotated rx 43.39 ry 15.84 rz 65.61 deg; joints [-0.239, -10.397, 78.376, 155.644, 94.401, 23.993, 178.286]
  MoveL 429 to (27.34, -59.87, -164.55) mm, rotated rx 43.39 ry 15.84 rz 65.61 deg; joints [-0.244, -10.384, 78.371, 155.64, 94.409, 23.992, 178.286]
  MoveL 430 to (27.3, -60, -164.67) mm, rotated rx 43.39 ry 15.84 rz 65.61 deg; joints [-0.245, -10.373, 78.348, 155.639, 94.398, 23.997, 178.286]
  MoveL 431 to (27.19, -60.38, -164.69) mm, rotated rx 43.39 ry 15.84 rz 65.61 deg; joints [-0.242, -10.363, 78.309, 155.643, 94.371, 24.008, 178.286]
  MoveL 432 to (27.06, -60.83, -164.7) mm, rotated rx 43.39 ry 15.84 rz 65.61 deg; joints [-0.239, -10.352, 78.265, 155.646, 94.34, 24.021, 178.286]
  MoveL 433 to (26.65, -62.35, -164.7) mm, rotated rx 43.39 ry 15.84 rz 65.61 deg; joints [-0.23, -10.318, 78.116, 155.659, 94.234, 24.065, 178.286]
  MoveL 434 to (26.5, -62.88, -164.72) mm, rotated rx 43.39 ry 15.84 rz 65.61 deg; joints [-0.226, -10.305, 78.063, 155.663, 94.197, 24.08, 178.286]
  MoveL 435 to (26.32, -63.4, -164.77) mm, rotated rx 43.39 ry 15.84 rz 65.61 deg; joints [-0.222, -10.289, 78.006, 155.668, 94.16, 24.096, 178.286]
  MoveL 436 to (26.12, -63.94, -164.85) mm, rotated rx 43.39 ry 15.84 rz 65.61 deg; joints [-0.218, -10.27, 77.946, 155.673, 94.121, 24.112, 178.286]
  MoveL 437 to (25.94, -64.46, -164.91) mm, rotated rx 43.39 ry 15.84 rz 65.61 deg; joints [-0.214, -10.253, 77.888, 155.677, 94.083, 24.127, 178.286]
  MoveL 438 to (25.79, -64.97, -164.93) mm, rotated rx 43.39 ry 15.84 rz 65.61 deg; joints [-0.211, -10.239, 77.836, 155.682, 94.047, 24.142, 178.286]
  MoveL 439 to (25.65, -65.45, -164.95) mm, rotated rx 43.39 ry 15.84 rz 65.61 deg; joints [-0.208, -10.227, 77.787, 155.685, 94.014, 24.156, 178.286]
  MoveL 440 to (25.5, -65.88, -165) mm, rotated rx 43.39 ry 15.84 rz 65.61 deg; joints [-0.205, -10.213, 77.74, 155.689, 93.983, 24.168, 178.286]
  MoveL 441 to (25.36, -66.3, -165.03) mm, rotated rx 43.39 ry 15.84 rz 65.61 deg; joints [-0.201, -10.201, 77.695, 155.693, 93.953, 24.181, 178.286]
  MoveL 442 to (25.22, -66.78, -165.05) mm, rotated rx 43.39 ry 15.84 rz 65.61 deg; joints [-0.198, -10.188, 77.646, 155.697, 93.919, 24.195, 178.286]
  MoveL 443 to (25.05, -67.34, -165.07) mm, rotated rx 43.39 ry 15.84 rz 65.61 deg; joints [-0.195, -10.174, 77.589, 155.702, 93.88, 24.211, 178.286]
  MoveL 444 to (24.83, -68.01, -165.12) mm, rotated rx 43.39 ry 15.84 rz 65.61 deg; joints [-0.19, -10.154, 77.517, 155.707, 93.832, 24.23, 178.286]
  MoveL 445 to (24.66, -68.59, -165.15) mm, rotated rx 43.39 ry 15.84 rz 65.61 deg; joints [-0.186, -10.138, 77.457, 155.712, 93.791, 24.247, 178.286]
  MoveL 446 to (24.11, -70.62, -165.15) mm, rotated rx 43.39 ry 15.84 rz 65.61 deg; joints [-0.173, -10.091, 77.256, 155.728, 93.649, 24.306, 178.286]
  MoveL 447 to (23.08, -73.34, -165.48) mm, rotated rx 43.39 ry 15.84 rz 65.61 deg; joints [-0.15, -9.997, 76.949, 155.753, 93.451, 24.386, 178.286]
  MoveL 448 to (22.41, -74.45, -165.9) mm, rotated rx 43.39 ry 15.84 rz 65.61 deg; joints [-0.137, -9.933, 76.793, 155.768, 93.364, 24.419, 178.286]
  MoveL 449 to (21.64, -75.39, -166.47) mm, rotated rx 43.39 ry 15.84 rz 65.61 deg; joints [-0.122, -9.858, 76.635, 155.783, 93.287, 24.447, 178.286]
  MoveL 450 to (19.78, -76.75, -168.12) mm, rotated rx 43.39 ry 15.84 rz 65.61 deg; joints [-0.087, -9.675, 76.316, 155.818, 93.156, 24.491, 178.286]
  MoveL 451 to (17.5, -77.42, -170.43) mm, rotated rx 43.39 ry 15.84 rz 65.61 deg; joints [-0.045, -9.447, 75.989, 155.858, 93.06, 24.516, 178.286]
  MoveL 452 to (15.47, -77.35, -172.74) mm, rotated rx 43.39 ry 15.84 rz 65.61 deg; joints [-0.01, -9.238, 75.739, 155.89, 93.016, 24.52, 178.286]
  MoveL 453 to (14.81, -77.01, -173.64) mm, rotated rx 43.39 ry 15.84 rz 65.61 deg; joints [0, -9.165, 75.674, 155.899, 93.022, 24.513, 178.286]
  MoveL 454 to (14.37, -76.46, -174.38) mm, rotated rx 43.39 ry 15.84 rz 65.61 deg; joints [0.006, -9.113, 75.649, 155.904, 93.046, 24.5, 178.286]
  MoveL 455 to (14.24, -76.11, -174.69) mm, rotated rx 43.39 ry 15.84 rz 65.61 deg; joints [0.007, -9.095, 75.652, 155.904, 93.065, 24.491, 178.286]
  MoveL 456 to (14.17, -75.71, -174.96) mm, rotated rx 43.39 ry 15.84 rz 65.61 deg; joints [0.007, -9.082, 75.665, 155.903, 93.089, 24.481, 178.286]
  MoveL 457 to (14.19, -74.75, -175.37) mm, rotated rx 43.39 ry 15.84 rz 65.61 deg; joints [0.003, -9.071, 75.72, 155.898, 93.15, 24.455, 178.286]
  MoveL 458 to (14.45, -73.59, -175.62) mm, rotated rx 43.39 ry 15.84 rz 65.61 deg; joints [-0.006, -9.081, 75.816, 155.889, 93.229, 24.423, 178.286]
  MoveL 459 to (14.94, -72.22, -175.7) mm, rotated rx 43.39 ry 15.84 rz 65.61 deg; joints [-0.019, -9.112, 75.952, 155.874, 93.327, 24.385, 178.286]
  MoveL 460 to (16.33, -68.83, -175.7) mm, rotated rx 43.39 ry 15.84 rz 65.61 deg; joints [-0.056, -9.206, 76.31, 155.835, 93.574, 24.29, 178.286]
  MoveL 461 to (16.52, -68.41, -175.69) mm, rotated rx 43.39 ry 15.84 rz 65.61 deg; joints [-0.06, -9.219, 76.356, 155.83, 93.605, 24.278, 178.286]
  MoveL 462 to (16.69, -68.04, -175.66) mm, rotated rx 43.39 ry 15.84 rz 65.61 deg; joints [-0.065, -9.232, 76.398, 155.825, 93.632, 24.267, 178.286]
  MoveL 463 to (16.88, -67.6, -175.64) mm, rotated rx 43.39 ry 15.84 rz 65.61 deg; joints [-0.07, -9.245, 76.446, 155.82, 93.664, 24.255, 178.286]
  MoveL 464 to (18.27, -64.21, -175.64) mm, rotated rx 43.39 ry 15.84 rz 65.61 deg; joints [-0.106, -9.338, 76.801, 155.779, 93.91, 24.16, 178.286]
  MoveL 465 to (18.5, -63.72, -175.62) mm, rotated rx 43.39 ry 15.84 rz 65.61 deg; joints [-0.112, -9.353, 76.855, 155.773, 93.946, 24.146, 178.286]
  MoveL 466 to (18.76, -63.24, -175.59) mm, rotated rx 43.39 ry 15.84 rz 65.61 deg; joints [-0.119, -9.37, 76.91, 155.766, 93.982, 24.133, 178.286]
  MoveL 467 to (19.03, -62.83, -175.54) mm, rotated rx 43.39 ry 15.84 rz 65.61 deg; joints [-0.126, -9.387, 76.96, 155.759, 94.013, 24.122, 178.286]
  MoveL 468 to (19.27, -62.53, -175.48) mm, rotated rx 43.39 ry 15.84 rz 65.61 deg; joints [-0.132, -9.402, 77.001, 155.752, 94.037, 24.113, 178.286]
  MoveL 469 to (19.41, -62.41, -175.31) mm, rotated rx 43.39 ry 15.84 rz 65.61 deg; joints [-0.134, -9.419, 77.03, 155.75, 94.049, 24.109, 178.286]
  MoveL 470 to (19.45, -62.42, -174.98) mm, rotated rx 43.39 ry 15.84 rz 65.61 deg; joints [-0.131, -9.442, 77.056, 155.753, 94.051, 24.107, 178.286]
  MoveL 471 to (19.37, -62.55, -174.47) mm, rotated rx 43.39 ry 15.84 rz 65.61 deg; joints [-0.123, -9.471, 77.08, 155.761, 94.045, 24.106, 178.286]
  MoveL 472 to (20.19, -62.67, -173.01) mm, rotated rx 43.39 ry 15.84 rz 65.61 deg; joints [-0.13, -9.588, 77.213, 155.753, 94.061, 24.102, 178.286]
  MoveL 473 to (23.74, -60.3, -173.01) mm, rotated rx 43.39 ry 15.84 rz 65.61 deg; joints [-0.24, -9.723, 77.556, 155.649, 94.268, 24.054, 178.286]
  MoveL 474 to (25.44, -59.17, -172.96) mm, rotated rx 43.39 ry 15.84 rz 65.61 deg; joints [-0.292, -9.79, 77.722, 155.599, 94.366, 24.031, 178.286]
  MoveL 475 to (27.08, -58.08, -172.88) mm, rotated rx 43.39 ry 15.84 rz 65.61 deg; joints [-0.341, -9.857, 77.886, 155.551, 94.462, 24.008, 178.286]
  MoveL 476 to (28.76, -56.96, -172.79) mm, rotated rx 43.39 ry 15.84 rz 65.61 deg; joints [-0.392, -9.925, 78.052, 155.502, 94.559, 23.984, 178.286]
  MoveL 477 to (30.4, -55.86, -172.69) mm, rotated rx 43.39 ry 15.84 rz 65.61 deg; joints [-0.442, -9.993, 78.216, 155.454, 94.654, 23.961, 178.286]
  MoveL 478 to (32.15, -54.72, -172.65) mm, rotated rx 43.39 ry 15.84 rz 65.61 deg; joints [-0.496, -10.06, 78.382, 155.401, 94.753, 23.938, 178.286]
  MoveL 479 to (34.04, -53.59, -172.62) mm, rotated rx 43.39 ry 15.84 rz 65.61 deg; joints [-0.555, -10.13, 78.552, 155.345, 94.853, 23.916, 178.286]
  MoveL 480 to (36.07, -52.12, -172.45) mm, rotated rx 43.39 ry 15.84 rz 65.61 deg; joints [-0.616, -10.217, 78.766, 155.286, 94.977, 23.883, 178.286]
  MoveL 481 to (37.93, -50.87, -172.2) mm, rotated rx 43.39 ry 15.84 rz 65.61 deg; joints [-0.671, -10.301, 78.96, 155.232, 95.085, 23.856, 178.286]
  MoveL 482 to (39.75, -49.65, -172.07) mm, rotated rx 43.39 ry 15.84 rz 65.61 deg; joints [-0.726, -10.376, 79.14, 155.178, 95.189, 23.829, 178.286]
  MoveL 483 to (41.52, -48.46, -171.83) mm, rotated rx 43.39 ry 15.84 rz 65.61 deg; joints [-0.779, -10.456, 79.324, 155.127, 95.291, 23.803, 178.286]
  MoveL 484 to (43.29, -47.27, -171.71) mm, rotated rx 43.39 ry 15.84 rz 65.61 deg; joints [-0.833, -10.528, 79.499, 155.074, 95.393, 23.777, 178.286]
  MoveL 485 to (45.06, -46.07, -171.59) mm, rotated rx 43.39 ry 15.84 rz 65.61 deg; joints [-0.887, -10.6, 79.673, 155.021, 95.494, 23.752, 178.286]
  MoveL 486 to (46.82, -44.87, -171.35) mm, rotated rx 43.39 ry 15.84 rz 65.61 deg; joints [-0.94, -10.679, 79.856, 154.969, 95.596, 23.724, 178.286]
  MoveL 487 to (48.59, -43.67, -171.23) mm, rotated rx 43.39 ry 15.84 rz 65.61 deg; joints [-0.994, -10.75, 80.029, 154.916, 95.697, 23.698, 178.286]
  MoveL 488 to (50.35, -42.46, -171.11) mm, rotated rx 43.39 ry 15.84 rz 65.61 deg; joints [-1.048, -10.82, 80.201, 154.862, 95.797, 23.672, 178.286]
  MoveL 489 to (52.11, -41.26, -171) mm, rotated rx 43.39 ry 15.84 rz 65.61 deg; joints [-1.102, -10.89, 80.373, 154.809, 95.897, 23.646, 178.286]
  MoveL 490 to (53.86, -40.04, -170.77) mm, rotated rx 43.39 ry 15.84 rz 65.61 deg; joints [-1.155, -10.967, 80.554, 154.757, 95.999, 23.618, 178.286]
  MoveL 491 to (55.62, -38.83, -170.66) mm, rotated rx 43.39 ry 15.84 rz 65.61 deg; joints [-1.21, -11.036, 80.725, 154.703, 96.099, 23.592, 178.286]
  MoveL 492 to (57.07, -37.78, -170.4) mm, rotated rx 43.39 ry 15.84 rz 65.61 deg; joints [-1.252, -11.104, 80.882, 154.66, 96.186, 23.567, 178.286]
  MoveL 493 to (58.4, -36.8, -170.08) mm, rotated rx 43.39 ry 15.84 rz 65.61 deg; joints [-1.29, -11.173, 81.034, 154.622, 96.267, 23.543, 178.286]
  MoveL 494 to (59.64, -35.84, -169.66) mm, rotated rx 43.39 ry 15.84 rz 65.61 deg; joints [-1.325, -11.244, 81.188, 154.587, 96.346, 23.518, 178.286]
  MoveL 495 to (57.93, -36.14, -168.71) mm, rotated rx 43.39 ry 15.84 rz 65.61 deg; joints [-1.256, -11.258, 81.176, 154.65, 96.314, 23.508, 178.286]
  MoveL 496 to (58.48, -35.82, -168.58) mm, rotated rx 43.39 ry 15.84 rz 65.61 deg; joints [-1.272, -11.284, 81.231, 154.635, 96.341, 23.501, 178.286]
  MoveL 497 to (59.01, -35.59, -168.49) mm, rotated rx 43.39 ry 15.84 rz 65.61 deg; joints [-1.288, -11.307, 81.275, 154.619, 96.363, 23.496, 178.286]
  MoveL 498 to (59.54, -35.47, -168.46) mm, rotated rx 43.39 ry 15.84 rz 65.61 deg; joints [-1.305, -11.325, 81.305, 154.603, 96.377, 23.496, 178.286]
  MoveL 499 to (60.07, -35.41, -168.44) mm, rotated rx 43.39 ry 15.84 rz 65.61 deg; joints [-1.322, -11.34, 81.329, 154.587, 96.387, 23.498, 178.286]
  MoveL 500 to (63.75, -35.39, -168.43) mm, rotated rx 43.39 ry 15.84 rz 65.61 deg; joints [-1.444, -11.438, 81.456, 154.475, 96.431, 23.523, 178.286]
  MoveL 501 to (64.21, -35.38, -168.42) mm, rotated rx 43.39 ry 15.84 rz 65.61 deg; joints [-1.459, -11.452, 81.473, 154.461, 96.437, 23.526, 178.286]
  MoveL 502 to (64.63, -35.36, -168.39) mm, rotated rx 43.39 ry 15.84 rz 65.61 deg; joints [-1.473, -11.465, 81.491, 154.449, 96.443, 23.528, 178.286]
  MoveL 503 to (65.11, -35.35, -168.38) mm, rotated rx 43.39 ry 15.84 rz 65.61 deg; joints [-1.489, -11.478, 81.508, 154.434, 96.449, 23.532, 178.286]
  MoveL 504 to (65.64, -35.35, -168.38) mm, rotated rx 43.39 ry 15.84 rz 65.61 deg; joints [-1.506, -11.492, 81.526, 154.418, 96.455, 23.535, 178.286]
  MoveL 505 to (67.21, -35.35, -168.38) mm, rotated rx 43.39 ry 15.84 rz 65.61 deg; joints [-1.559, -11.533, 81.579, 154.37, 96.473, 23.547, 178.286]
  MoveL 506 to (67.84, -35.33, -168.36) mm, rotated rx 43.39 ry 15.84 rz 65.61 deg; joints [-1.579, -11.551, 81.602, 154.351, 96.481, 23.551, 178.286]
  MoveL 507 to (68.55, -35.3, -168.32) mm, rotated rx 43.39 ry 15.84 rz 65.61 deg; joints [-1.602, -11.573, 81.631, 154.33, 96.491, 23.555, 178.286]
  MoveL 508 to (69.2, -35.29, -168.3) mm, rotated rx 43.39 ry 15.84 rz 65.61 deg; joints [-1.624, -11.591, 81.656, 154.31, 96.5, 23.559, 178.286]
  MoveL 509 to (70.25, -35.29, -168.3) mm, rotated rx 43.39 ry 15.84 rz 65.61 deg; joints [-1.658, -11.619, 81.69, 154.278, 96.512, 23.566, 178.286]
  MoveL 510 to (71.69, -35.36, -168.39) mm, rotated rx 43.39 ry 15.84 rz 65.61 deg; joints [-1.708, -11.65, 81.726, 154.233, 96.523, 23.58, 178.286]
  MoveL 511 to (72.86, -35.57, -168.64) mm, rotated rx 43.39 ry 15.84 rz 65.61 deg; joints [-1.75, -11.662, 81.729, 154.195, 96.521, 23.597, 178.286]
  MoveL 512 to (73.75, -35.91, -169.06) mm, rotated rx 43.39 ry 15.84 rz 65.61 deg; joints [-1.786, -11.654, 81.698, 154.164, 96.506, 23.618, 178.286]
  MoveL 513 to (74.09, -36.14, -169.33) mm, rotated rx 43.39 ry 15.84 rz 65.61 deg; joints [-1.801, -11.642, 81.67, 154.151, 96.493, 23.629, 178.286]
  MoveL 514 to (74.36, -36.4, -169.65) mm, rotated rx 43.39 ry 15.84 rz 65.61 deg; joints [-1.815, -11.626, 81.634, 154.14, 96.478, 23.642, 178.286]
  MoveL 515 to (74.68, -37.02, -170.4) mm, rotated rx 43.39 ry 15.84 rz 65.61 deg; joints [-1.836, -11.578, 81.537, 154.123, 96.437, 23.671, 178.286]
  MoveL 516 to (74.73, -37.78, -171.33) mm, rotated rx 43.39 ry 15.84 rz 65.61 deg; joints [-1.851, -11.51, 81.406, 154.113, 96.382, 23.703, 178.286]
  MoveL 517 to (73.99, -39.71, -173.68) mm, rotated rx 43.39 ry 15.84 rz 65.61 deg; joints [-1.86, -11.313, 81.044, 154.113, 96.235, 23.778, 178.286]
  MoveL 518 to (72.46, -41.6, -176.03) mm, rotated rx 43.39 ry 15.84 rz 65.61 deg; joints [-1.843, -11.096, 80.658, 154.136, 96.08, 23.847, 178.286]
  MoveL 519 to (70.46, -42.83, -177.71) mm, rotated rx 43.39 ry 15.84 rz 65.61 deg; joints [-1.8, -10.918, 80.361, 154.18, 95.966, 23.886, 178.286]
  MoveL 520 to (69.29, -43.19, -178.3) mm, rotated rx 43.39 ry 15.84 rz 65.61 deg; joints [-1.77, -10.845, 80.246, 154.209, 95.925, 23.894, 178.286]
  MoveL 521 to (68, -43.4, -178.72) mm, rotated rx 43.39 ry 15.84 rz 65.61 deg; joints [-1.733, -10.781, 80.154, 154.244, 95.894, 23.895, 178.286]
  MoveL 522 to (65.09, -43.32, -179.06) mm, rotated rx 43.39 ry 15.84 rz 65.61 deg; joints [-1.641, -10.683, 80.037, 154.328, 95.863, 23.873, 178.286]
  MoveL 523 to (61.97, -42.91, -179.06) mm, rotated rx 43.39 ry 15.84 rz 65.61 deg; joints [-1.537, -10.605, 79.966, 154.421, 95.852, 23.838, 178.286]
  MoveL 524 to (60.99, -42.84, -179.1) mm, rotated rx 43.39 ry 15.84 rz 65.61 deg; joints [-1.505, -10.577, 79.935, 154.45, 95.845, 23.829, 178.286]
  MoveL 525 to (60.47, -42.77, -179.1) mm, rotated rx 43.39 ry 15.84 rz 65.61 deg; joints [-1.488, -10.564, 79.923, 154.466, 95.843, 23.823, 178.286]
  MoveL 526 to (59.94, -42.7, -179.11) mm, rotated rx 43.39 ry 15.84 rz 65.61 deg; joints [-1.47, -10.551, 79.91, 154.482, 95.841, 23.817, 178.286]
  MoveL 527 to (59.37, -42.64, -179.13) mm, rotated rx 43.39 ry 15.84 rz 65.61 deg; joints [-1.452, -10.535, 79.894, 154.499, 95.838, 23.811, 178.286]
  MoveL 528 to (58.73, -42.6, -179.19) mm, rotated rx 43.39 ry 15.84 rz 65.61 deg; joints [-1.431, -10.514, 79.871, 154.517, 95.833, 23.805, 178.286]
  MoveL 529 to (58.15, -42.54, -179.22) mm, rotated rx 43.39 ry 15.84 rz 65.61 deg; joints [-1.412, -10.498, 79.854, 154.534, 95.829, 23.8, 178.286]
  MoveL 530 to (57.63, -42.48, -179.23) mm, rotated rx 43.39 ry 15.84 rz 65.61 deg; joints [-1.395, -10.484, 79.84, 154.55, 95.827, 23.794, 178.286]
  MoveL 531 to (57.15, -42.45, -179.26) mm, rotated rx 43.39 ry 15.84 rz 65.61 deg; joints [-1.38, -10.469, 79.824, 154.564, 95.823, 23.79, 178.286]
  MoveL 532 to (56.7, -42.42, -179.31) mm, rotated rx 43.39 ry 15.84 rz 65.61 deg; joints [-1.366, -10.454, 79.807, 154.577, 95.819, 23.786, 178.286]
  MoveL 533 to (56.24, -42.39, -179.35) mm, rotated rx 43.39 ry 15.84 rz 65.61 deg; joints [-1.351, -10.44, 79.791, 154.59, 95.815, 23.782, 178.286]
  MoveL 534 to (55.73, -42.33, -179.36) mm, rotated rx 43.39 ry 15.84 rz 65.61 deg; joints [-1.334, -10.427, 79.777, 154.605, 95.812, 23.777, 178.286]
  MoveL 535 to (55.23, -42.28, -179.37) mm, rotated rx 43.39 ry 15.84 rz 65.61 deg; joints [-1.317, -10.413, 79.764, 154.62, 95.81, 23.772, 178.286]
  MoveL 536 to (54.71, -42.25, -179.38) mm, rotated rx 43.39 ry 15.84 rz 65.61 deg; joints [-1.3, -10.4, 79.748, 154.636, 95.805, 23.767, 178.286]
  MoveL 537 to (54.22, -42.28, -179.39) mm, rotated rx 43.39 ry 15.84 rz 65.61 deg; joints [-1.284, -10.385, 79.727, 154.65, 95.798, 23.765, 178.286]
  MoveL 538 to (53.75, -42.36, -179.42) mm, rotated rx 43.39 ry 15.84 rz 65.61 deg; joints [-1.27, -10.369, 79.702, 154.664, 95.786, 23.764, 178.286]
  MoveL 539 to (53.32, -42.5, -179.47) mm, rotated rx 43.39 ry 15.84 rz 65.61 deg; joints [-1.256, -10.353, 79.671, 154.677, 95.772, 23.766, 178.286]
  MoveL 540 to (52.89, -42.67, -179.52) mm, rotated rx 43.39 ry 15.84 rz 65.61 deg; joints [-1.243, -10.336, 79.639, 154.69, 95.755, 23.769, 178.286]
  MoveL 541 to (54.38, -42.34, -180.48) mm, rotated rx 43.39 ry 15.84 rz 65.61 deg; joints [-1.304, -10.317, 79.645, 154.633, 95.787, 23.777, 178.286]
  MoveL 542 to (52.93, -43.26, -180.86) mm, rotated rx 43.39 ry 15.84 rz 65.61 deg; joints [-1.263, -10.242, 79.487, 154.674, 95.707, 23.799, 178.286]
  MoveL 543 to (51.36, -44.17, -181.14) mm, rotated rx 43.39 ry 15.84 rz 65.61 deg; joints [-1.216, -10.169, 79.334, 154.719, 95.626, 23.819, 178.286]
  MoveL 544 to (49.66, -45.1, -181.34) mm, rotated rx 43.39 ry 15.84 rz 65.61 deg; joints [-1.165, -10.098, 79.178, 154.77, 95.543, 23.838, 178.286]
  MoveL 545 to (47.77, -46.1, -181.56) mm, rotated rx 43.39 ry 15.84 rz 65.61 deg; joints [-1.107, -10.019, 79.009, 154.825, 95.452, 23.858, 178.286]
  MoveL 546 to (45.87, -47.07, -181.68) mm, rotated rx 43.39 ry 15.84 rz 65.61 deg; joints [-1.048, -9.947, 78.85, 154.882, 95.364, 23.877, 178.286]
  MoveL 547 to (43.96, -48.04, -181.79) mm, rotated rx 43.39 ry 15.84 rz 65.61 deg; joints [-0.989, -9.875, 78.69, 154.939, 95.275, 23.895, 178.286]
  MoveL 548 to (42.07, -49.02, -182.02) mm, rotated rx 43.39 ry 15.84 rz 65.61 deg; joints [-0.932, -9.795, 78.519, 154.994, 95.184, 23.914, 178.286]
  MoveL 549 to (40.16, -49.98, -182.14) mm, rotated rx 43.39 ry 15.84 rz 65.61 deg; joints [-0.873, -9.722, 78.358, 155.051, 95.096, 23.932, 178.286]
  MoveL 550 to (38.25, -50.95, -182.26) mm, rotated rx 43.39 ry 15.84 rz 65.61 deg; joints [-0.814, -9.649, 78.197, 155.107, 95.007, 23.95, 178.286]
  MoveL 551 to (36.35, -51.91, -182.5) mm, rotated rx 43.39 ry 15.84 rz 65.61 deg; joints [-0.757, -9.568, 78.026, 155.162, 94.916, 23.969, 178.286]
  MoveL 552 to (34.44, -52.87, -182.62) mm, rotated rx 43.39 ry 15.84 rz 65.61 deg; joints [-0.698, -9.494, 77.864, 155.218, 94.827, 23.986, 178.286]
  MoveL 553 to (32.53, -53.82, -182.74) mm, rotated rx 43.39 ry 15.84 rz 65.61 deg; joints [-0.639, -9.42, 77.701, 155.274, 94.737, 24.004, 178.286]
  MoveL 554 to (30.73, -54.71, -182.93) mm, rotated rx 43.39 ry 15.84 rz 65.61 deg; joints [-0.585, -9.345, 77.541, 155.326, 94.652, 24.02, 178.286]
  MoveL 555 to (29.09, -55.52, -183.15) mm, rotated rx 43.39 ry 15.84 rz 65.61 deg; joints [-0.536, -9.274, 77.393, 155.373, 94.574, 24.036, 178.286]
  MoveL 556 to (27.33, -56.39, -183.25) mm, rotated rx 43.39 ry 15.84 rz 65.61 deg; joints [-0.482, -9.205, 77.243, 155.424, 94.492, 24.052, 178.286]
  MoveL 557 to (25.43, -57.45, -183.25) mm, rotated rx 43.39 ry 15.84 rz 65.61 deg; joints [-0.422, -9.137, 77.079, 155.481, 94.396, 24.071, 178.286]
  MoveL 558 to (22.98, -58.64, -183.34) mm, rotated rx 43.39 ry 15.84 rz 65.61 deg; joints [-0.347, -9.045, 76.876, 155.552, 94.282, 24.092, 178.286]
  MoveL 559 to (20.72, -59.62, -183.58) mm, rotated rx 43.39 ry 15.84 rz 65.61 deg; joints [-0.279, -8.952, 76.685, 155.616, 94.183, 24.109, 178.286]
  MoveL 560 to (18.89, -60.5, -183.76) mm, rotated rx 43.39 ry 15.84 rz 65.61 deg; joints [-0.224, -8.875, 76.523, 155.668, 94.096, 24.125, 178.286]
  MoveL 561 to (17.2, -61.3, -184.08) mm, rotated rx 43.39 ry 15.84 rz 65.61 deg; joints [-0.175, -8.794, 76.362, 155.714, 94.016, 24.141, 178.286]
  MoveL 562 to (15.35, -62.18, -184.26) mm, rotated rx 43.39 ry 15.84 rz 65.61 deg; joints [-0.12, -8.717, 76.199, 155.767, 93.929, 24.157, 178.286]
  MoveL 563 to (13.57, -63.02, -184.46) mm, rotated rx 43.39 ry 15.84 rz 65.61 deg; joints [-0.067, -8.64, 76.04, 155.817, 93.845, 24.173, 178.286]
  MoveL 564 to (11.81, -63.81, -184.74) mm, rotated rx 43.39 ry 15.84 rz 65.61 deg; joints [-0.016, -8.56, 75.879, 155.865, 93.764, 24.187, 178.286]
  MoveL 565 to (10.91, -63.64, -185.51) mm, rotated rx 43.39 ry 15.84 rz 65.61 deg; joints [0.003, -8.486, 75.799, 155.882, 93.755, 24.183, 178.286]
  MoveL 566 to (11.12, -63.33, -185.89) mm, rotated rx 43.39 ry 15.84 rz 65.61 deg; joints [-0.008, -8.471, 75.804, 155.872, 93.775, 24.179, 178.286]
  MoveL 567 to (11.14, -63.25, -186.14) mm, rotated rx 43.39 ry 15.84 rz 65.61 deg; joints [-0.011, -8.457, 75.793, 155.869, 93.779, 24.179, 178.286]
  MoveL 568 to (10.99, -63.4, -186.26) mm, rotated rx 43.39 ry 15.84 rz 65.61 deg; joints [-0.008, -8.442, 75.764, 155.871, 93.765, 24.184, 178.286]
  MoveL 569 to (10.68, -63.82, -186.31) mm, rotated rx 43.39 ry 15.84 rz 65.61 deg; joints [0, -8.424, 75.71, 155.88, 93.732, 24.195, 178.286]
  MoveL 570 to (10.31, -64.38, -186.35) mm, rotated rx 43.39 ry 15.84 rz 65.61 deg; joints [0.01, -8.402, 75.643, 155.89, 93.689, 24.21, 178.286]
  MoveL 571 to (9.53, -65.74, -186.35) mm, rotated rx 43.39 ry 15.84 rz 65.61 deg; joints [0.032, -8.358, 75.49, 155.912, 93.586, 24.247, 178.286]
  MoveL 572 to (9.26, -66.21, -186.36) mm, rotated rx 43.39 ry 15.84 rz 65.61 deg; joints [0.039, -8.342, 75.436, 155.92, 93.55, 24.26, 178.286]
  MoveL 573 to (8.97, -66.67, -186.38) mm, rotated rx 43.39 ry 15.84 rz 65.61 deg; joints [0.047, -8.325, 75.382, 155.928, 93.515, 24.272, 178.286]
  MoveL 574 to (8.67, -67.13, -186.43) mm, rotated rx 43.39 ry 15.84 rz 65.61 deg; joints [0.055, -8.306, 75.325, 155.936, 93.479, 24.285, 178.286]
  MoveL 575 to (8.35, -67.59, -186.5) mm, rotated rx 43.39 ry 15.84 rz 65.61 deg; joints [0.063, -8.284, 75.266, 155.944, 93.443, 24.298, 178.286]
  MoveL 576 to (8.04, -68.04, -186.56) mm, rotated rx 43.39 ry 15.84 rz 65.61 deg; joints [0.071, -8.264, 75.208, 155.953, 93.407, 24.31, 178.286]
  MoveL 577 to (7.78, -68.47, -186.58) mm, rotated rx 43.39 ry 15.84 rz 65.61 deg; joints [0.078, -8.248, 75.157, 155.96, 93.375, 24.322, 178.286]
  MoveL 578 to (7.55, -68.86, -186.6) mm, rotated rx 43.39 ry 15.84 rz 65.61 deg; joints [0.084, -8.234, 75.111, 155.966, 93.345, 24.332, 178.286]
  MoveL 579 to (6.77, -70.22, -186.6) mm, rotated rx 43.39 ry 15.84 rz 65.61 deg; joints [0.106, -8.189, 74.957, 155.988, 93.241, 24.369, 178.286]
  MoveL 580 to (6.5, -70.67, -186.61) mm, rotated rx 43.39 ry 15.84 rz 65.61 deg; joints [0.113, -8.173, 74.905, 155.996, 93.207, 24.381, 178.286]
  MoveL 581 to (6.25, -71.07, -186.64) mm, rotated rx 43.39 ry 15.84 rz 65.61 deg; joints [0.12, -8.157, 74.856, 156.002, 93.176, 24.392, 178.286]
  MoveL 582 to (6, -71.44, -186.69) mm, rotated rx 43.39 ry 15.84 rz 65.61 deg; joints [0.127, -8.141, 74.809, 156.009, 93.147, 24.403, 178.286]
  MoveL 583 to (5.75, -71.82, -186.73) mm, rotated rx 43.39 ry 15.84 rz 65.61 deg; joints [0.133, -8.125, 74.761, 156.016, 93.117, 24.413, 178.286]
  MoveL 584 to (5.49, -72.24, -186.74) mm, rotated rx 43.39 ry 15.84 rz 65.61 deg; joints [0.14, -8.11, 74.712, 156.022, 93.085, 24.424, 178.286]
  MoveL 585 to (5.23, -72.69, -186.74) mm, rotated rx 43.39 ry 15.84 rz 65.61 deg; joints [0.147, -8.094, 74.66, 156.03, 93.05, 24.437, 178.286]
  MoveL 586 to (3.53, -75.08, -187.08) mm, rotated rx 43.39 ry 15.84 rz 65.61 deg; joints [0.191, -7.982, 74.347, 156.073, 92.859, 24.502, 178.286]
  MoveL 587 to (2.59, -75.99, -187.5) mm, rotated rx 43.39 ry 15.84 rz 65.61 deg; joints [0.214, -7.911, 74.192, 156.095, 92.779, 24.528, 178.286]
  MoveL 588 to (1.58, -76.72, -188.09) mm, rotated rx 43.39 ry 15.84 rz 65.61 deg; joints [0.236, -7.83, 74.037, 156.117, 92.708, 24.55, 178.286]
  MoveL 589 to (-0.63, -77.63, -189.78) mm, rotated rx 43.39 ry 15.84 rz 65.61 deg; joints [0.282, -7.637, 73.729, 156.16, 92.595, 24.579, 178.286]
  MoveL 590 to (-3.09, -77.79, -192.14) mm, rotated rx 43.39 ry 15.84 rz 65.61 deg; joints [0.33, -7.405, 73.424, 156.204, 92.521, 24.591, 178.286]
  MoveL 591 to (-5.11, -77.28, -194.51) mm, rotated rx 43.39 ry 15.84 rz 65.61 deg; joints [0.365, -7.196, 73.195, 156.236, 92.497, 24.586, 178.286]
  MoveL 592 to (-5.7, -76.82, -195.43) mm, rotated rx 43.39 ry 15.84 rz 65.61 deg; joints [0.373, -7.124, 73.139, 156.243, 92.509, 24.577, 178.286]
  MoveL 593 to (-6.01, -76.2, -196.19) mm, rotated rx 43.39 ry 15.84 rz 65.61 deg; joints [0.374, -7.075, 73.121, 156.244, 92.538, 24.564, 178.286]
  MoveL 594 to (-6.06, -75.84, -196.51) mm, rotated rx 43.39 ry 15.84 rz 65.61 deg; joints [0.372, -7.059, 73.127, 156.242, 92.558, 24.555, 178.286]
  MoveL 595 to (-6.04, -75.44, -196.78) mm, rotated rx 43.39 ry 15.84 rz 65.61 deg; joints [0.369, -7.048, 73.142, 156.238, 92.583, 24.546, 178.286]
  MoveL 596 to (-5.79, -74.54, -197.21) mm, rotated rx 43.39 ry 15.84 rz 65.61 deg; joints [0.358, -7.043, 73.202, 156.227, 92.644, 24.524, 178.286]
  MoveL 597 to (-5.25, -73.49, -197.46) mm, rotated rx 43.39 ry 15.84 rz 65.61 deg; joints [0.34, -7.06, 73.3, 156.21, 92.721, 24.498, 178.286]
  MoveL 598 to (-4.43, -72.3, -197.54) mm, rotated rx 43.39 ry 15.84 rz 65.61 deg; joints [0.316, -7.098, 73.436, 156.186, 92.814, 24.467, 178.286]
  MoveL 599 to (-3.49, -71.04, -197.54) mm, rotated rx 43.39 ry 15.84 rz 65.61 deg; joints [0.289, -7.148, 73.59, 156.16, 92.915, 24.435, 178.286]
  MoveL 600 to (-3.16, -70.63, -197.54) mm, rotated rx 43.39 ry 15.84 rz 65.61 deg; joints [0.28, -7.164, 73.642, 156.151, 92.948, 24.424, 178.286]
  MoveL 601 to (-2.8, -70.18, -197.51) mm, rotated rx 43.39 ry 15.84 rz 65.61 deg; joints [0.27, -7.185, 73.701, 156.141, 92.985, 24.412, 178.286]
  MoveL 602 to (-2.37, -69.7, -197.44) mm, rotated rx 43.39 ry 15.84 rz 65.61 deg; joints [0.259, -7.21, 73.768, 156.13, 93.025, 24.399, 178.286]
  MoveL 603 to (-2.01, -69.26, -197.42) mm, rotated rx 43.39 ry 15.84 rz 65.61 deg; joints [0.249, -7.229, 73.824, 156.12, 93.06, 24.388, 178.286]
  MoveL 604 to (-1.69, -68.84, -197.41) mm, rotated rx 43.39 ry 15.84 rz 65.61 deg; joints [0.24, -7.246, 73.876, 156.111, 93.094, 24.377, 178.286]
  MoveL 605 to (-1.37, -68.43, -197.4) mm, rotated rx 43.39 ry 15.84 rz 65.61 deg; joints [0.23, -7.263, 73.927, 156.102, 93.127, 24.366, 178.286]
  MoveL 606 to (-1.04, -68.04, -197.36) mm, rotated rx 43.39 ry 15.84 rz 65.61 deg; joints [0.221, -7.282, 73.98, 156.093, 93.159, 24.356, 178.286]
  MoveL 607 to (-0.7, -67.68, -197.28) mm, rotated rx 43.39 ry 15.84 rz 65.61 deg; joints [0.212, -7.303, 74.033, 156.085, 93.19, 24.346, 178.286]
  MoveL 608 to (-0.34, -67.31, -197.18) mm, rotated rx 43.39 ry 15.84 rz 65.61 deg; joints [0.203, -7.326, 74.088, 156.076, 93.221, 24.336, 178.286]
  MoveL 609 to (0, -66.94, -197.11) mm, rotated rx 43.39 ry 15.84 rz 65.61 deg; joints [0.194, -7.347, 74.142, 156.067, 93.252, 24.326, 178.286]
  MoveL 610 to (0.34, -66.53, -197.08) mm, rotated rx 43.39 ry 15.84 rz 65.61 deg; joints [0.185, -7.365, 74.196, 156.057, 93.286, 24.315, 178.286]
  MoveL 611 to (0.66, -66.12, -197.07) mm, rotated rx 43.39 ry 15.84 rz 65.61 deg; joints [0.176, -7.382, 74.247, 156.048, 93.319, 24.305, 178.286]
  MoveL 612 to (2.23, -64.1, -197.06) mm, rotated rx 43.39 ry 15.84 rz 65.61 deg; joints [0.13, -7.461, 74.493, 156.004, 93.479, 24.253, 178.286]
  MoveL 613 to (2.51, -63.83, -197.04) mm, rotated rx 43.39 ry 15.84 rz 65.61 deg; joints [0.122, -7.475, 74.531, 155.996, 93.502, 24.246, 178.286]
  MoveL 614 to (2.65, -63.74, -196.92) mm, rotated rx 43.39 ry 15.84 rz 65.61 deg; joints [0.12, -7.488, 74.554, 155.993, 93.511, 24.243, 178.286]
  MoveL 615 to (2.59, -63.8, -196.69) mm, rotated rx 43.39 ry 15.84 rz 65.61 deg; joints [0.124, -7.501, 74.564, 155.998, 93.509, 24.242, 178.286]
  MoveL 616 to (2.3, -64.02, -196.33) mm, rotated rx 43.39 ry 15.84 rz 65.61 deg; joints [0.138, -7.513, 74.563, 156.01, 93.493, 24.243, 178.286]
  MoveL 617 to (3.05, -64.21, -195.59) mm, rotated rx 43.39 ry 15.84 rz 65.61 deg; joints [0.123, -7.581, 74.635, 155.997, 93.5, 24.247, 178.286]
  MoveL 618 to (5.06, -63.52, -195.57) mm, rotated rx 43.39 ry 15.84 rz 65.61 deg; joints [0.06, -7.651, 74.778, 155.938, 93.577, 24.239, 178.286]
  MoveL 619 to (7.13, -62.84, -195.44) mm, rotated rx 43.39 ry 15.84 rz 65.61 deg; joints [-0.003, -7.729, 74.932, 155.879, 93.656, 24.231, 178.286]
  MoveL 620 to (9.3, -62.16, -195.18) mm, rotated rx 43.39 ry 15.84 rz 65.61 deg; joints [-0.068, -7.819, 75.1, 155.819, 93.737, 24.222, 178.286]
  MoveL 621 to (11.31, -61.51, -195.05) mm, rotated rx 43.39 ry 15.84 rz 65.61 deg; joints [-0.13, -7.896, 75.248, 155.762, 93.812, 24.214, 178.286]
  MoveL 622 to (13.26, -60.88, -194.79) mm, rotated rx 43.39 ry 15.84 rz 65.61 deg; joints [-0.187, -7.978, 75.401, 155.708, 93.886, 24.205, 178.286]
  MoveL 623 to (15.27, -60.24, -194.43) mm, rotated rx 43.39 ry 15.84 rz 65.61 deg; joints [-0.246, -8.068, 75.565, 155.653, 93.962, 24.195, 178.286]
  MoveL 624 to (17.3, -59.56, -194.3) mm, rotated rx 43.39 ry 15.84 rz 65.61 deg; joints [-0.309, -8.145, 75.715, 155.594, 94.039, 24.187, 178.286]
  MoveL 625 to (19.31, -58.88, -194.2) mm, rotated rx 43.39 ry 15.84 rz 65.61 deg; joints [-0.371, -8.219, 75.861, 155.537, 94.114, 24.178, 178.286]
  MoveL 626 to (21.34, -58.18, -194.05) mm, rotated rx 43.39 ry 15.84 rz 65.61 deg; joints [-0.433, -8.296, 76.012, 155.478, 94.191, 24.169, 178.286]
  MoveL 627 to (23.33, -57.54, -193.76) mm, rotated rx 43.39 ry 15.84 rz 65.61 deg; joints [-0.492, -8.38, 76.167, 155.423, 94.265, 24.16, 178.286]
  MoveL 628 to (25.38, -56.79, -193.42) mm, rotated rx 43.39 ry 15.84 rz 65.61 deg; joints [-0.553, -8.471, 76.338, 155.366, 94.347, 24.148, 178.286]
  MoveL 629 to (27.38, -56.09, -193.24) mm, rotated rx 43.39 ry 15.84 rz 65.61 deg; joints [-0.614, -8.55, 76.49, 155.308, 94.424, 24.138, 178.286]
  MoveL 630 to (29.41, -55.38, -193.13) mm, rotated rx 43.39 ry 15.84 rz 65.61 deg; joints [-0.677, -8.623, 76.637, 155.249, 94.5, 24.129, 178.286]
  MoveL 631 to (31.41, -54.68, -193.06) mm, rotated rx 43.39 ry 15.84 rz 65.61 deg; joints [-0.74, -8.694, 76.779, 155.19, 94.575, 24.12, 178.286]
  MoveL 632 to (33.43, -53.95, -192.83) mm, rotated rx 43.39 ry 15.84 rz 65.61 deg; joints [-0.801, -8.775, 76.935, 155.133, 94.653, 24.109, 178.286]
  MoveL 633 to (35.43, -53.24, -192.7) mm, rotated rx 43.39 ry 15.84 rz 65.61 deg; joints [-0.863, -8.849, 77.082, 155.074, 94.728, 24.099, 178.286]
  MoveL 634 to (37.45, -52.53, -192.62) mm, rotated rx 43.39 ry 15.84 rz 65.61 deg; joints [-0.926, -8.92, 77.225, 155.014, 94.803, 24.09, 178.286]
  MoveL 635 to (39.44, -51.79, -192.39) mm, rotated rx 43.39 ry 15.84 rz 65.61 deg; joints [-0.987, -9, 77.38, 154.957, 94.88, 24.079, 178.286]
  MoveL 636 to (41.46, -51.04, -192.16) mm, rotated rx 43.39 ry 15.84 rz 65.61 deg; joints [-1.048, -9.082, 77.537, 154.899, 94.959, 24.067, 178.286]
  MoveL 637 to (43.51, -50.29, -192.01) mm, rotated rx 43.39 ry 15.84 rz 65.61 deg; joints [-1.112, -9.158, 77.688, 154.839, 95.036, 24.057, 178.286]
  MoveL 638 to (45.26, -49.62, -191.89) mm, rotated rx 43.39 ry 15.84 rz 65.61 deg; joints [-1.167, -9.223, 77.819, 154.787, 95.105, 24.046, 178.286]
  MoveL 639 to (46.77, -48.98, -191.68) mm, rotated rx 43.39 ry 15.84 rz 65.61 deg; joints [-1.212, -9.287, 77.946, 154.744, 95.168, 24.035, 178.286]
  MoveL 640 to (48.06, -48.34, -191.35) mm, rotated rx 43.39 ry 15.84 rz 65.61 deg; joints [-1.249, -9.352, 78.072, 154.708, 95.229, 24.021, 178.286]
  MoveL 641 to (46.61, -48.61, -190.4) mm, rotated rx 43.39 ry 15.84 rz 65.61 deg; joints [-1.19, -9.372, 78.071, 154.763, 95.201, 24.01, 178.286]
  MoveL 642 to (47.08, -48.45, -190.4) mm, rotated rx 43.39 ry 15.84 rz 65.61 deg; joints [-1.205, -9.387, 78.102, 154.748, 95.218, 24.008, 178.286]
  MoveL 643 to (47.56, -48.32, -190.39) mm, rotated rx 43.39 ry 15.84 rz 65.61 deg; joints [-1.22, -9.402, 78.13, 154.734, 95.232, 24.008, 178.286]
  MoveL 644 to (48.09, -48.29, -190.37) mm, rotated rx 43.39 ry 15.84 rz 65.61 deg; joints [-1.237, -9.419, 78.154, 154.718, 95.242, 24.01, 178.286]
  MoveL 645 to (48.65, -48.31, -190.33) mm, rotated rx 43.39 ry 15.84 rz 65.61 deg; joints [-1.255, -9.436, 78.175, 154.702, 95.248, 24.014, 178.286]
  MoveL 646 to (49.26, -48.39, -190.27) mm, rotated rx 43.39 ry 15.84 rz 65.61 deg; joints [-1.274, -9.455, 78.195, 154.685, 95.251, 24.021, 178.286]
  MoveL 647 to (49.83, -48.5, -190.23) mm, rotated rx 43.39 ry 15.84 rz 65.61 deg; joints [-1.293, -9.472, 78.208, 154.668, 95.251, 24.028, 178.286]
  MoveL 648 to (50.38, -48.64, -190.21) mm, rotated rx 43.39 ry 15.84 rz 65.61 deg; joints [-1.311, -9.486, 78.217, 154.652, 95.249, 24.036, 178.286]
  MoveL 649 to (50.88, -48.77, -190.21) mm, rotated rx 43.39 ry 15.84 rz 65.61 deg; joints [-1.328, -9.497, 78.223, 154.637, 95.247, 24.044, 178.286]
  MoveL 650 to (51.39, -48.9, -190.21) mm, rotated rx 43.39 ry 15.84 rz 65.61 deg; joints [-1.344, -9.51, 78.23, 154.622, 95.245, 24.052, 178.286]
  MoveL 651 to (51.97, -49.02, -190.17) mm, rotated rx 43.39 ry 15.84 rz 65.61 deg; joints [-1.363, -9.527, 78.244, 154.605, 95.245, 24.059, 178.286]
  MoveL 652 to (52.62, -49.12, -190.08) mm, rotated rx 43.39 ry 15.84 rz 65.61 deg; joints [-1.383, -9.548, 78.265, 154.587, 95.247, 24.066, 178.286]
  MoveL 653 to (53.13, -49.23, -190.03) mm, rotated rx 43.39 ry 15.84 rz 65.61 deg; joints [-1.4, -9.564, 78.277, 154.573, 95.247, 24.073, 178.286]
